// TwinCAT 3 PLC project PLC1
// ProgramVersion: 3.1.4026.16
// CompilerDefines: VISU_USEPROPERTYINFO
// libraries:
//   SH_Light, * (StroemHansen)
//   Tc2_EnOcean, * (Beckhoff Automation GmbH)
//   Tc2_Standard, * (Beckhoff Automation GmbH)
//   Tc2_System, * (Beckhoff Automation GmbH)
//   Tc2_Utilities, * (Beckhoff Automation GmbH)
//   Tc3_DALI, * (Beckhoff Automation GmbH)
//   Tc3_System_DK, * (Beckhoff - DK)
//   VisuDialogs, * (System)
// project tree:
//   DUTs/DALI/ E_DALIExtendedFadeTime.TcTLEO (not stored), ST_DALI102Parameters.TcDUT (not stored), ST_DALI103Parameters.TcDUT (not stored), ST_DALIMemoryBank.TcDUT (not stored), ST_DALI_GrpAssignment.TcDUT (not stored), ST_GroupSort.TcDUT (not stored)
//   DUTs/EnOcean/ ST_ReadSAB05.TcDUT (not stored), ST_WriteSAB05.TcDUT (not stored)
//   / FastTask.TcTTO (not stored), GlobalTextList.TcGTLO (not stored), PlcTask.TcTTO (not stored), Visualization Manager.TcVMO (not stored)
//   GVLs/ GVL_AHDataModbus.TcGVL, GVL_EnOcean.TcGVL, GVL_Skalering.TcGVL
//   POUs/01_System/01_System/GVLs/ GVL_EtherCAT.TcGVL (not stored)
//   POUs/01_System/01_System/ P_SystemDK.TcPOU (not stored)
//   POUs/AHModbusComm/ P_AHModbusComm.TcPOU
//   POUs/Alle_Rum/Gange/Gang_3_109/ P_Gang_3_109_Kantine.TcPOU, Visualization_4_308.TcVIS (excluded from build)
//   POUs/Alle_Rum/Gange/Gang_4_208/ P_Gang_4_208.TcPOU, Visualization_5_338_1.TcVIS (excluded from build)
//   POUs/Alle_Rum/Gange/Gang_4_211/ P_Gang_4_211.TcPOU, Visualization_5_338_1_1_1_1.TcVIS (excluded from build)
//   POUs/Alle_Rum/Gange/Gang_4_210A/ P_Gang_4_210A.TcPOU, Visualization_4_307_1_1.TcVIS (excluded from build)
//   POUs/Alle_Rum/Rum_Med_DALI_Pir/Rum_4_206/ P_Rum_4_206.TcPOU, Visualization_5_338_1_1.TcVIS (excluded from build)
//   POUs/Alle_Rum/Rum_Med_DALI_Pir/Rum_4_211A/ P_Rum_4_211A.TcPOU, Visualization_5_338_1_1_1.TcVIS (excluded from build)
//   POUs/Alle_Rum/Rum_Med_DALI_Pir/Rum_4_207/ P_Rum_4_207.TcPOU, Visualization_4_307_1.TcVIS (excluded from build)
//   POUs/Alle_Rum/Rum_Med_DALI_Pir/Rum_4_213_Og_4_215_Foldedoer/ P_Foldedoer_4_213.TcPOU, P_Rum_4_213.TcPOU, P_Rum_4_215.TcPOU
//   POUs/Alle_Rum/Trapper/ P_DigTest.TcPOU
//   POUs/DALI/DALI_Setup/ DALI_Commissioning.TcPOU (not stored)
//   POUs/DALI/DALI_Setup/FBs/ FB_Part102Addressing.TcPOU (not stored), FB_Part102Commands.TcPOU (not stored), FB_Part102Groups.TcPOU (not stored), FB_Part102MemoryPages.TcPOU (not stored), FB_Part102Parameters.TcPOU (not stored), FB_Part102Scenes.TcPOU (not stored), FB_Part102SetFading.TcPOU (not stored), FB_Part103Addressing.TcPOU (not stored), FB_Part103MemoryPages.TcPOU (not stored), FB_Part103Identify.TcPOU (not stored), FB_Part103Parameters.TcPOU (not stored), FB_Part202Emergency.TcPOU (not stored), FB_Part205Incandescent.TcPOU (not stored), FB_Part207LED.TcPOU (not stored), FB_Part208Switching.TcPOU (not stored), FB_Part300GenericDevice.TcPOU (not stored), FB_Part301PushButton.TcPOU (not stored), FB_Part302AbsoluteInputDevice.TcPOU (not stored), FB_Part303OccupancySensor.TcPOU (not stored), FB_Part304LightSensor.TcPOU (not stored), GearType.TcPOU (not stored)
//   POUs/DALI/DALI_Setup/GVLs/ GVL_Internal.TcGVL (not stored)
//   POUs/DALI/DALI_Setup/VISUs/TextLists/ CommandOnTerminalEvent.TcTLO, DimmingCurve.TcTLO, EventPriority.TcTLO (not stored), EventScheme.TcTLO, ExtendedFadeTime.TcTLO (not stored), FadeRate.TcTLO (not stored), FadeTime.TcTLO, FastFadeTime.TcTLO (not stored), TextList_Dialogs.TcTLO (not stored)
//   POUs/DALI/DALI_Setup/VISUs/ Visu_DALICommissioning.TcVIS
//   POUs/DALI/DALI_Setup/VISUs/Visu_DALICommissioning/ Visu_KL6821Configuration.TcVIS (not stored) (excluded from build), Visu_Part102Addressing.TcVIS, Visu_Part102Commands.TcVIS (not stored), Visu_Part102Groups.TcVIS, Visu_Part102MemoryBank.TcVIS (not stored), Visu_Part102Parameters.TcVIS, Visu_Part102Scenes.TcVIS, Visu_Part102SetFading.TcVIS, Visu_Part103Addressing.TcVIS, Visu_Part103Identify.TcVIS (not stored), Visu_Part103MemoryBank.TcVIS (not stored), Visu_Part103Parameters.TcVIS (not stored), Visu_Part202.TcVIS (not stored), Visu_Part202Commands.TcVIS (not stored), Visu_Part202Parameters.TcVIS (not stored), Visu_Part202Status.TcVIS (not stored), Visu_Part205.TcVIS (not stored), Visu_Part205Parameters.TcVIS (not stored), Visu_Part205Status.TcVIS (not stored), Visu_Part207.TcVIS, Visu_Part207Parameters.TcVIS (not stored), Visu_Part207Status.TcVIS, Visu_Part208Switching.TcVIS (not stored), Visu_Part300GenericDevice.TcVIS, Visu_Part301PushButton.TcVIS (not stored), Visu_Part302AbsoluteInputDevice.TcVIS (not stored), Visu_Part303OccupancySensor.TcVIS, Visu_Part304LightSensor.TcVIS (not stored), Visu_Welcome.TcVIS (not stored)
//   POUs/DALI/PRGs/Background/ P_DALI_Background.TcPOU (not stored)
//   POUs/DALI/PRGs/Diag/ P_DALI_DIAG.TcPOU (not stored)
//   POUs/DALI/PRGs/EnergyData/ P_DALI_Energy_Firmware_Test.TcPOU (not stored) (excluded from build), P_DALI_Energy_Line.TcPOU (not stored)
//   POUs/EnOcean/ P_EnOcean.TcPOU
//   POUs/ MAIN.TcPOU
//   POUs/Tester/ P_DALI2_Test.TcPOU (not stored) (excluded from build), P_Test_TypeA.TcPOU (not stored) (excluded from build), Visualization.TcVIS (not stored) (excluded from build)
// real-time tasks:
//   TASK PlcTask: cycle T#40ms, priority 21, ADS port 350
//   TASK FastTask: cycle T#4ms, priority 20, ADS port 351
// I/O:
//   DEVICE Device 1 (Beckhoff CCAT)
//   DEVICE Device 3 (CX-BK)
//     Box 1 (CX-BK)
// variable links:
//   PLC1/PLC1 Instance <-> Device 3 (CX-BK)/Box 1 (CX-BK)
//     FastTask Inputs/P_DALI_Background.arrKL6821InData[1] @bit 16 <-> Term 4 (KL6821)/Channel 1/Data In 0
//     FastTask Inputs/P_DALI_Background.arrKL6821InData[1] @bit 24 <-> Term 4 (KL6821)/Channel 1/Data In 1
//     FastTask Inputs/P_DALI_Background.arrKL6821InData[1] @bit 32 <-> Term 4 (KL6821)/Channel 1/Data In 2
//     FastTask Inputs/P_DALI_Background.arrKL6821InData[1] @bit 40 <-> Term 4 (KL6821)/Channel 1/Data In 3
//     FastTask Inputs/P_DALI_Background.arrKL6821InData[2] @bit 16 <-> Term 5 (KL6821)/Channel 1/Data In 0
//     FastTask Inputs/P_DALI_Background.arrKL6821InData[2] @bit 24 <-> Term 5 (KL6821)/Channel 1/Data In 1
//     FastTask Inputs/P_DALI_Background.arrKL6821InData[2] @bit 32 <-> Term 5 (KL6821)/Channel 1/Data In 2
//     FastTask Inputs/P_DALI_Background.arrKL6821InData[2] @bit 40 <-> Term 5 (KL6821)/Channel 1/Data In 3
//     FastTask Inputs/P_DALI_Background.arrKL6821InData[3] @bit 16 <-> Term 6 (KL6821)/Channel 1/Data In 0
//     FastTask Inputs/P_DALI_Background.arrKL6821InData[3] @bit 24 <-> Term 6 (KL6821)/Channel 1/Data In 1
//     FastTask Inputs/P_DALI_Background.arrKL6821InData[3] @bit 32 <-> Term 6 (KL6821)/Channel 1/Data In 2
//     FastTask Inputs/P_DALI_Background.arrKL6821InData[3] @bit 40 <-> Term 6 (KL6821)/Channel 1/Data In 3
//     FastTask Inputs/P_DALI_Background.arrKL6821InData[1] <-> Term 4 (KL6821)/Channel 1/State
//     FastTask Inputs/P_DALI_Background.arrKL6821InData[2] <-> Term 5 (KL6821)/Channel 1/State
//     FastTask Inputs/P_DALI_Background.arrKL6821InData[3] <-> Term 6 (KL6821)/Channel 1/State
//     FastTask Inputs/P_EnOcean.stKL6581_in @bit 8 <-> Term 2 (KL6581)/Channel 1/Input CNODE
//     FastTask Inputs/P_EnOcean.stKL6581_in @bit {24..48 step 8} <-> Term 2 (KL6581)/Channel 1/Input DB{0..3}  (4 links)
//     FastTask Inputs/P_EnOcean.stKL6581_in @bit {56..80 step 8} <-> Term 2 (KL6581)/Channel 1/Input ID{0..3}  (4 links)
//     FastTask Inputs/P_EnOcean.stKL6581_in @bit 16 <-> Term 2 (KL6581)/Channel 1/Input ORG
//     FastTask Inputs/P_EnOcean.stKL6581_in @bit 88 <-> Term 2 (KL6581)/Channel 1/Input STATUS
//     FastTask Inputs/P_EnOcean.stKL6581_in <-> Term 2 (KL6581)/Channel 1/Status
//     FastTask Outputs/P_DALI_Background.arrKL6821OutData[1] <-> Term 4 (KL6821)/Channel 1/Ctrl
//     FastTask Outputs/P_DALI_Background.arrKL6821OutData[2] <-> Term 5 (KL6821)/Channel 1/Ctrl
//     FastTask Outputs/P_DALI_Background.arrKL6821OutData[3] <-> Term 6 (KL6821)/Channel 1/Ctrl
//     FastTask Outputs/P_DALI_Background.arrKL6821OutData[1] @bit 16 <-> Term 4 (KL6821)/Channel 1/Data Out 0
//     FastTask Outputs/P_DALI_Background.arrKL6821OutData[1] @bit 24 <-> Term 4 (KL6821)/Channel 1/Data Out 1
//     FastTask Outputs/P_DALI_Background.arrKL6821OutData[1] @bit 32 <-> Term 4 (KL6821)/Channel 1/Data Out 2
//     FastTask Outputs/P_DALI_Background.arrKL6821OutData[1] @bit 40 <-> Term 4 (KL6821)/Channel 1/Data Out 3
//     FastTask Outputs/P_DALI_Background.arrKL6821OutData[2] @bit 16 <-> Term 5 (KL6821)/Channel 1/Data Out 0
//     FastTask Outputs/P_DALI_Background.arrKL6821OutData[2] @bit 24 <-> Term 5 (KL6821)/Channel 1/Data Out 1
//     FastTask Outputs/P_DALI_Background.arrKL6821OutData[2] @bit 32 <-> Term 5 (KL6821)/Channel 1/Data Out 2
//     FastTask Outputs/P_DALI_Background.arrKL6821OutData[2] @bit 40 <-> Term 5 (KL6821)/Channel 1/Data Out 3
//     FastTask Outputs/P_DALI_Background.arrKL6821OutData[3] @bit 16 <-> Term 6 (KL6821)/Channel 1/Data Out 0
//     FastTask Outputs/P_DALI_Background.arrKL6821OutData[3] @bit 24 <-> Term 6 (KL6821)/Channel 1/Data Out 1
//     FastTask Outputs/P_DALI_Background.arrKL6821OutData[3] @bit 32 <-> Term 6 (KL6821)/Channel 1/Data Out 2
//     FastTask Outputs/P_DALI_Background.arrKL6821OutData[3] @bit 40 <-> Term 6 (KL6821)/Channel 1/Data Out 3
//     FastTask Outputs/P_EnOcean.stKL6581_out <-> Term 2 (KL6581)/Channel 1/Control
//     FastTask Outputs/P_EnOcean.stKL6581_out @bit 8 <-> Term 2 (KL6581)/Channel 1/Output CNODE
//     FastTask Outputs/P_EnOcean.stKL6581_out @bit {24..48 step 8} <-> Term 2 (KL6581)/Channel 1/Output DB{0..3}  (4 links)
//     FastTask Outputs/P_EnOcean.stKL6581_out @bit {56..80 step 8} <-> Term 2 (KL6581)/Channel 1/Output ID{0..3}  (4 links)
//     FastTask Outputs/P_EnOcean.stKL6581_out @bit 16 <-> Term 2 (KL6581)/Channel 1/Output ORG
//     FastTask Outputs/P_EnOcean.stKL6581_out @bit 88 <-> Term 2 (KL6581)/Channel 1/Output STATUS
//     PlcTask Inputs/MAIN.nCX8200_State <-> Inputs/State
//     PlcTask Inputs/P_Foldedoer_4_213.bFoldingDoorOpen <-> Term 3 (KL1408)/Channel 2/Input

// ---- GVLs/GVL_AHDataModbus.TcGVL
{attribute 'qualified_only'}
VAR_GLOBAL
//AH pir data out
	nAH_NeighborRoomsPir_Out		    AT %MB600	: UINT;
	
//AH pir data in
	arrAH_NeighborRoomsPir_In								: ARRAY[1..byNumberOfAH_Neighbors] OF UINT;
	arrAH_NeighborRoomsPir										: ARRAY[1..byNumberOfAH_Neighbors] OF ARRAY[0..15] OF BOOL;
	
//Schneider data out
	nCX8200_State_MB					AT %MB1000		: UINT;
	arrFB_DALIDiagErrorId			(*AT %MW1002*)	: ARRAY[1..SH_Light.DALI_Param.MAX_DALIV2_LINES] OF UDINT;
	arrKL6821InDataStatus				AT %MB1014		: ARRAY[1..SH_Light.DALI_Param.MAX_DALIV2_LINES] OF WORD;
	arrDALILineShrtAddrErr				AT %MB1026		: ARRAY[1..SH_Light.DALI_Param.MAX_DALIV2_LINES] OF UINT;
	EnOceanError						AT %MB1038		: UINT;
	nTotalEnergy10kWh						AT %MB1040		: UINT;
	nMaxControlGearOperatingHours 	    AT %MB1042		: UINT;
		uiPirOffDelayTimeAllRooms_MB   AT %MB1044   : UINT := 30;
END_VAR
VAR_GLOBAL CONSTANT
	byNumberOfAH_Neighbors									: BYTE := 25;
END_VAR

// ---- GVLs/GVL_EnOcean.TcGVL
{attribute 'qualified_only'}
VAR_GLOBAL
//Atrium
	strEnOceanSwitch_Gang_3_109_PladeA				: Tc2_EnOcean.STR_EnOceanSwitch;
	strEnOceanSwitch_AtriumNiveau_PladeB				: Tc2_EnOcean.STR_EnOceanSwitch;
	strEnOceanSwitch_AtriumNiveau_Service				: Tc2_EnOcean.STR_EnOceanSwitch;	

	//Gange
    strEnOceanSwitch_Gang_4_211_Indgang				: Tc2_EnOcean.STR_EnOceanSwitch;
	strEnOceanSwitch_Gang_4_211_Ekstra					: Tc2_EnOcean.STR_EnOceanSwitch;
	
	//Rum				
	strEnOceanSwitch_Rum_4_206_Indgang				: Tc2_EnOcean.STR_EnOceanSwitch;
	strEnOceanSwitch_Rum_4_206_Ekstra					: Tc2_EnOcean.STR_EnOceanSwitch;
	
	strEnOceanSwitch_Rum_4_207_Indgang				: Tc2_EnOcean.STR_EnOceanSwitch;
	strEnOceanSwitch_Rum_4_207_Ekstra					: Tc2_EnOcean.STR_EnOceanSwitch;
	
	strEnOceanSwitch_Rum_4_211A_Indgang				: Tc2_EnOcean.STR_EnOceanSwitch;
	strEnOceanSwitch_Rum_4_211A_Ekstra				: Tc2_EnOcean.STR_EnOceanSwitch;
	
	strEnOceanSwitch_Rum_4_213_Indgang				: Tc2_EnOcean.STR_EnOceanSwitch;
	strEnOceanSwitch_Rum_4_213_Pendler				: Tc2_EnOcean.STR_EnOceanSwitch;
	
	strEnOceanSwitch_Rum_4_215								: Tc2_EnOcean.STR_EnOceanSwitch;
	
END_VAR

// ---- GVLs/GVL_Skalering.TcGVL
//{attribute 'qualified_only'}
VAR_GLOBAL
rMeassure_Zone1 :REAL:= 604; 
rRead_Zone1     :REAL:= 340;

rMeassure_Zone2 :REAL:=611;
rRead_Zone2     :REAL:=374;

rMeassure_Zone3 :REAL:=986;
rRead_Zone3     :REAL:=524;

rMeassure_Zone4 :REAL:=770;
rRead_Zone4     :REAL:=506;

rMeassure_Zone5 :REAL:=734;
rRead_Zone5     :REAL:=395;

rMeassure_Zone6 :REAL:=890;
rRead_Zone6     :REAL:=476;

rMeassure_Zone7 :REAL:=710;
rRead_Zone7     :REAL:=654;

rMeassure_Zone8 :REAL:=604;
rRead_Zone8     :REAL:=292;

rMeassure_Zone9 :REAL:=572;
rRead_Zone9     :REAL:=348;

rMeassure_Zone10:REAL:= 790;
rRead_Zone10    :REAL:=434;

rMeassure_Zone11 :REAL:=691;
rRead_Zone11     :REAL:=426;

END_VAR

// ---- POUs/AHModbusComm/P_AHModbusComm.TcPOU
PROGRAM P_AHModbusComm
VAR
	arrfbReadAHPirData		: ARRAY[1..GVL_AHDataModbus.byNumberOfAH_Neighbors] OF SH_Light.FB_ReadAHPirData;
	arrReadAHPirData			: ARRAY[1..GVL_AHDataModbus.byNumberOfAH_Neighbors] OF BOOL;
	
	arrfbTriggerPulses			: ARRAY[1..GVL_AHDataModbus.byNumberOfAH_Neighbors] OF SH_Light.FB_ClockPulse;
	arrGeneratePulses			: ARRAY[1..GVL_AHDataModbus.byNumberOfAH_Neighbors] OF BOOL := [GVL_AHDataModbus.byNumberOfAH_Neighbors(TRUE)];
	tTimeInterval					: TIME := T#1S;
	tPulseTime					: TIME := T#1S;
	
	byLineId						: BYTE;
	byAHId							: BYTE;
	
			
	fbWritePirDelayTime		: R_TRIG;
	bRunOverrideOnce		: BOOL := FALSE;
	bEnableDelayTimeOverride : BOOL := FALSE;
	uiPirOffDelayTimeAllRooms : UINT := 30;
END_VAR

VAR CONSTANT
	arrstNeighborIPAddr					: ARRAY[1..GVL_AHDataModbus.byNumberOfAH_Neighbors] OF SH_Light.ST_NeighborIP := [
																								(sIP := '172.24.195.161', IsNeighbor := FALSE),
																							    (sIP := '172.24.195.162', IsNeighbor := FALSE), // AH1-2
																								(sIP := '172.24.195.163', IsNeighbor := FALSE), 
																							(sIP := '172.24.195.164', IsNeighbor := TRUE), 
																							(sIP := '172.24.195.165', IsNeighbor := TRUE), 
																								(sIP := '172.24.195.166', IsNeighbor := FALSE), 
																								(sIP := '172.24.195.167', IsNeighbor := FALSE), 
																								(sIP := '172.24.195.168', IsNeighbor := FALSE), 
																							(sIP := '172.24.195.169', IsNeighbor := TRUE), // AH3-2
																								(sIP := '172.24.195.170', IsNeighbor := FALSE), 
																								(sIP := '172.24.195.171', IsNeighbor := FALSE), 
																								(sIP := '172.24.195.172', IsNeighbor := FALSE), 
																								(sIP := '172.24.195.173', IsNeighbor := FALSE), 
																							(sIP := '172.24.195.174', IsNeighbor := TRUE), 
																								(sIP := '172.24.195.175', IsNeighbor := FALSE), 
																								(sIP := '172.24.195.176', IsNeighbor := FALSE), 
																								(sIP := '172.24.195.177', IsNeighbor := FALSE),
																							(sIP := '172.24.195.178', IsNeighbor := TRUE),
																							(sIP := '172.24.195.179', IsNeighbor := TRUE), // AH5-2
																								(sIP := '172.24.195.180', IsNeighbor := FALSE),
																								(sIP := '172.24.195.181', IsNeighbor := FALSE),
																								(sIP := '172.24.195.182', IsNeighbor := FALSE),
																								(sIP := '172.24.195.183', IsNeighbor := FALSE),
																								(sIP := '172.24.195.184', IsNeighbor := FALSE),
																								(sIP := '172.24.195.185', IsNeighbor := FALSE)];
	arrMBAddr					: ARRAY[1..GVL_AHDataModbus.byNumberOfAH_Neighbors] OF WORD := [GVL_AHDataModbus.byNumberOfAH_Neighbors(12588)]; //modbus-adresser
END_VAR

A_AHNeighborRoomsPirIn();
A_AHNeighborRoomsPirOut();
A_DALILineShrtAddrErr();
A_DelayTimeAllRooms();

ACTION A_AHNeighborRoomsPirIn:
FOR byAHId := 1 TO GVL_AHDataModbus.byNumberOfAH_Neighbors DO
//Generate Pulses
	arrfbTriggerPulses[byAHId](bGenerateClockPulses:= arrGeneratePulses[byAHId], tTimeInterval:= tTimeInterval, tPulseTime:= tPulseTime);
	arrReadAHPirData[byAHId]:= arrfbTriggerPulses[byAHId].bPulse;
//Read data
	IF arrstNeighborIPAddr[byAHId].IsNeighbor THEN
	arrfbReadAHPirData[byAHId](	bReadAHPirData			:=	arrReadAHPirData[byAHId],
													sIPAddr							:=	arrstNeighborIPAddr[byAHId].sIP,
													nMBAddr						:=	arrMBAddr[byAHId],
													nMBDataBuffer				:=	GVL_AHDataModbus.arrAH_NeighborRoomsPir_In[byAHId],
													arrAH_NeighborRoomsPir	=>GVL_AHDataModbus.arrAH_NeighborRoomsPir[byAHId]);
	END_IF
END_FOR
END_ACTION

ACTION A_AHNeighborRoomsPirOut:
GVL_AHDataModbus.nAH_NeighborRoomsPir_Out.0		:= P_Gang_3_109_Kantine.bPirActive_MB;
GVL_AHDataModbus.nAH_NeighborRoomsPir_Out.1		:= P_Gang_4_208.bPirActive_MB;
//GVL_AHDataModbus.nAH_NeighborRoomsPir_Out.2		:=
//GVL_AHDataModbus.nAH_NeighborRoomsPir_Out.3		:=
//GVL_AHDataModbus.nAH_NeighborRoomsPir_Out.4		:= 
//GVL_AHDataModbus.nAH_NeighborRoomsPir_Out.5		:= 
//GVL_AHDataModbus.nAH_NeighborRoomsPir_Out.6		:=
//GVL_AHDataModbus.nAH_NeighborRoomsPir_Out.7		:= 
//GVL_AHDataModbus.nAH_NeighborRoomsPir_Out.8		:=
//GVL_AHDataModbus.nAH_NeighborRoomsPir_Out.9		:= 
//GVL_AHDataModbus.nAH_NeighborRoomsPir_Out.10	:
//GVL_AHDataModbus.nAH_NeighborRoomsPir_Out.11	:= 
//GVL_AHDataModbus.nAH_NeighborRoomsPir_Out.12	:=
//GVL_AHDataModbus.nAH_NeighborRoomsPir_Out.13	:=
END_ACTION

ACTION A_DALILineShrtAddrErr:
FOR  byLineId := 1 TO SH_Light.DALI_Param.MAX_DALIV2_LINES DO
	GVL_AHDataModbus.arrDALILineShrtAddrErr[byLineId] :=  TO_UINT(SH_Light.GVL_DALI_LatestError.arrLineShrtAddr[byLineId]);
END_FOR
END_ACTION

ACTION A_DelayTimeAllRooms:

fbWritePirDelayTime(CLK := GVL_AHDataModbus.uiPirOffDelayTimeAllRooms_MB<>uiPirOffDelayTimeAllRooms);

IF fbWritePirDelayTime.Q THEN
	bRunOverrideOnce := TRUE;
	bEnableDelayTimeOverride := TRUE;
	
//Indsæt kode
P_Gang_3_109_Kantine.fbWritePirDelayTIme(bEnableOverride := bEnableDelayTimeOverride, nOverRideValue := GVL_AHDataModbus.uiPirOffDelayTimeAllRooms_MB, nValIn1 := GVL_AHDataModbus.uiPirOffDelayTimeAllRooms_MB, nValIn2 := uiPirOffDelayTimeAllRooms);
P_Gang_4_208.fbWritePirDelayTIme(bEnableOverride := bEnableDelayTimeOverride, nOverRideValue := GVL_AHDataModbus.uiPirOffDelayTimeAllRooms_MB, nValIn1 := GVL_AHDataModbus.uiPirOffDelayTimeAllRooms_MB, nValIn2 := uiPirOffDelayTimeAllRooms);
P_Rum_4_206.fbWritePirDelayTIme(bEnableOverride := bEnableDelayTimeOverride, nOverRideValue := GVL_AHDataModbus.uiPirOffDelayTimeAllRooms_MB, nValIn1 := GVL_AHDataModbus.uiPirOffDelayTimeAllRooms_MB, nValIn2 := uiPirOffDelayTimeAllRooms);
P_Rum_4_207.fbWritePirDelayTIme(bEnableOverride := bEnableDelayTimeOverride, nOverRideValue := GVL_AHDataModbus.uiPirOffDelayTimeAllRooms_MB, nValIn1 := GVL_AHDataModbus.uiPirOffDelayTimeAllRooms_MB, nValIn2 := uiPirOffDelayTimeAllRooms);
P_Rum_4_211A.fbWritePirDelayTIme(bEnableOverride := bEnableDelayTimeOverride, nOverRideValue := GVL_AHDataModbus.uiPirOffDelayTimeAllRooms_MB, nValIn1 := GVL_AHDataModbus.uiPirOffDelayTimeAllRooms_MB, nValIn2 := uiPirOffDelayTimeAllRooms);
P_Rum_4_213.fbWritePirDelayTIme(bEnableOverride := bEnableDelayTimeOverride, nOverRideValue := GVL_AHDataModbus.uiPirOffDelayTimeAllRooms_MB, nValIn1 := GVL_AHDataModbus.uiPirOffDelayTimeAllRooms_MB, nValIn2 := uiPirOffDelayTimeAllRooms);
P_Gang_4_211.fbWritePirDelayTIme(bEnableOverride := bEnableDelayTimeOverride, nOverRideValue := GVL_AHDataModbus.uiPirOffDelayTimeAllRooms_MB, nValIn1 := GVL_AHDataModbus.uiPirOffDelayTimeAllRooms_MB, nValIn2 := uiPirOffDelayTimeAllRooms);
P_Rum_4_215.fbWritePirDelayTIme(bEnableOverride := bEnableDelayTimeOverride, nOverRideValue := GVL_AHDataModbus.uiPirOffDelayTimeAllRooms_MB, nValIn1 := GVL_AHDataModbus.uiPirOffDelayTimeAllRooms_MB, nValIn2 := uiPirOffDelayTimeAllRooms);ELSE
	IF bRunOverrideOnce THEN
		bEnableDelayTimeOverride := FALSE;
		
		//Indsæt kode
P_Gang_3_109_Kantine.fbWritePirDelayTIme(bEnableOverride := bEnableDelayTimeOverride, nOverRideValue := GVL_AHDataModbus.uiPirOffDelayTimeAllRooms_MB, nValIn1 := GVL_AHDataModbus.uiPirOffDelayTimeAllRooms_MB, nValIn2 := uiPirOffDelayTimeAllRooms);
P_Gang_4_208.fbWritePirDelayTIme(bEnableOverride := bEnableDelayTimeOverride, nOverRideValue := GVL_AHDataModbus.uiPirOffDelayTimeAllRooms_MB, nValIn1 := GVL_AHDataModbus.uiPirOffDelayTimeAllRooms_MB, nValIn2 := uiPirOffDelayTimeAllRooms);
P_Rum_4_206.fbWritePirDelayTIme(bEnableOverride := bEnableDelayTimeOverride, nOverRideValue := GVL_AHDataModbus.uiPirOffDelayTimeAllRooms_MB, nValIn1 := GVL_AHDataModbus.uiPirOffDelayTimeAllRooms_MB, nValIn2 := uiPirOffDelayTimeAllRooms);
P_Rum_4_207.fbWritePirDelayTIme(bEnableOverride := bEnableDelayTimeOverride, nOverRideValue := GVL_AHDataModbus.uiPirOffDelayTimeAllRooms_MB, nValIn1 := GVL_AHDataModbus.uiPirOffDelayTimeAllRooms_MB, nValIn2 := uiPirOffDelayTimeAllRooms);
P_Rum_4_211A.fbWritePirDelayTIme(bEnableOverride := bEnableDelayTimeOverride, nOverRideValue := GVL_AHDataModbus.uiPirOffDelayTimeAllRooms_MB, nValIn1 := GVL_AHDataModbus.uiPirOffDelayTimeAllRooms_MB, nValIn2 := uiPirOffDelayTimeAllRooms);
P_Rum_4_213.fbWritePirDelayTIme(bEnableOverride := bEnableDelayTimeOverride, nOverRideValue := GVL_AHDataModbus.uiPirOffDelayTimeAllRooms_MB, nValIn1 := GVL_AHDataModbus.uiPirOffDelayTimeAllRooms_MB, nValIn2 := uiPirOffDelayTimeAllRooms);
P_Gang_4_211.fbWritePirDelayTIme(bEnableOverride := bEnableDelayTimeOverride, nOverRideValue := GVL_AHDataModbus.uiPirOffDelayTimeAllRooms_MB, nValIn1 := GVL_AHDataModbus.uiPirOffDelayTimeAllRooms_MB, nValIn2 := uiPirOffDelayTimeAllRooms);
P_Rum_4_215.fbWritePirDelayTIme(bEnableOverride := bEnableDelayTimeOverride, nOverRideValue := GVL_AHDataModbus.uiPirOffDelayTimeAllRooms_MB, nValIn1 := GVL_AHDataModbus.uiPirOffDelayTimeAllRooms_MB, nValIn2 := uiPirOffDelayTimeAllRooms);



bRunOverrideOnce := FALSE;
	END_IF
END_IF
END_ACTION

END_PROGRAM

// ---- POUs/Alle_Rum/Gange/Gang_3_109/P_Gang_3_109_Kantine.TcPOU
PROGRAM P_Gang_3_109_Kantine
VAR
(*Gangen består af to lysgrupper - 5 og 14 - på to forskellige DALI-linjer - 2 og 1 henh..
Begge grupper afhænger af samme PIR-input - pir-adr. 6, 7, 8, 9 og 10 - på DALI-linje 2.
Derfor oprettes to adskilte reguleringer med samme PV. Dvs., at knapfunktion og pirfunktion forbliver den samme.

En anden del af af hele gangen styres fra AH4_3. De to dele nabostyres med PIR-signaler over modbus-kommunikation*)

	arrfbLysGruppe			: ARRAY [1..2] OF FB_Light_Type_B;
	arrstDaliSetupGruppe	: ARRAY[1..2] OF SH_Light.ST_DALI_RoomSetup := 
	
													[(	byShrtAdr_Prim := 26, 
														byGrpAdr_Prim := 6, 
														eMod_Prim := E_DALIAddressType.Group, 
														//byShrtAdr_Sec := 1, 
														//byGrpAdr_Sec := 1, 
														//eMod_Sec := E_DALIAddressType.Short, 
														//byShrtAdr_Supl := 1, 
														DALI_LINE_NUM_PRIM := arrDALI_LINE_NUM_LIGHT[1], 
														DALI_LINE_NUM_SEC := 0, //0 = ingen zonestyring/vinduerække
														DALI_LINE_NUM_SUPL := arrDALI_LINE_NUM_PENDANTS[1]),
														
													(	byShrtAdr_Prim := 31, 
														byGrpAdr_Prim := 6, 
														eMod_Prim := E_DALIAddressType.Group, 
														//byShrtAdr_Sec := 1, 
														//byGrpAdr_Sec := 1, 
														//eMod_Sec := E_DALIAddressType.Short, 
														//byShrtAdr_Supl := 1, 
														DALI_LINE_NUM_PRIM := arrDALI_LINE_NUM_LIGHT[2], 
														DALI_LINE_NUM_SEC := 0, 
														DALI_LINE_NUM_SUPL := arrDALI_LINE_NUM_PENDANTS[2])];
														
	arrstLiveDataGruppe		: ARRAY [1..2] OF SH_Light.ST_LiveData;
	//stLiveData AT %MB22	: SH_Light.ST_LiveData;
	
	arrRunTuningGruppe: ARRAY[1..2] OF BOOL;
	
	
	
	bTopButtonZone1			: BOOL;
	bTopButtonZone1_Visu	: BOOL;
	bBottomButtonZone1		: BOOL;
	bBottomButtonZone1_Visu	: BOOL;
	bButtonZone2			: BOOL;
	bNeighborRoomsPir		: BOOL;
	fLuxOn					: REAL;
	fLuxDim					: REAL;
	tPIRDim					: TIME;
	tPIROff					: TIME;
	fOffsetSec				: REAL := 20;
	bOccupiedRoom			: BOOL;

	bRunTuning				: BOOL;
	


// Sensor Settings
	//fbSensor					: SH_Light.FB_NIKO_P46xx_1Pcs;
	fbSensor					: SH_Light.FB_NIKO_P46xx_3Pcs;
	//bySensorAddr				: BYTE := 17;
	arrSensorAddr				: ARRAY[1..3] OF BYTE := [3,4,5];
	bInitialize					: BOOL := TRUE;
	stDaliSensorSetup			: ST_DALI_NIKOP46SetupData;
	//bInitErr					: BOOL;
	//bInitDone					: BOOL;
	arrInitErr					: ARRAY [1..3] OF BOOL;
	arrInitDone					: ARRAY [1..3] OF BOOL;
	arrSensorScales				: ARRAY [1..10] OF SH_Light.ST_DALI_SensorScaleMode := [	(fMeassureMaxSensor := rMeassure_Zone11, fReadMaxSensor := rRead_Zone11),
																							(fMeassureMaxSensor := rMeassure_Zone11, fReadMaxSensor := rRead_Zone11),
																							(fMeassureMaxSensor := rMeassure_Zone11, fReadMaxSensor := rRead_Zone11),																					
																						7(())];
	bCancelHoldTimerOccupancy	: BOOL;
(*	eEventPriorityOccupancy		: E_DALIEventPriority := E_DALIEVENTPRIORITY.Middle;
	nHoldTimerOccupancy			: WORD := 5; // Value in s. 	
	nReportTimerOccupancy		: BYTE := 120; // Value in s, Preset manufacturer value
	nDeadtimeTimerOccupancy		: WORD := 100; // Value in ms, Predefined Value of DALI Standard
	bCancelHoldTimerOccupancy	: BOOL;
	nSensitivityOccupancy		: BYTE:= 3; //setting Sensivity (0..4) 0 (Off), 1 (Min), 2(Low), 3(High) and 4 (Max)

	bEnableLuxEvent				: BOOL;
	eEventPriorityBrightness	: E_DALIEventPriority := E_DALIEVENTPRIORITY.Middle;
	nDeadtimeTimerBrightness	: WORD := 1500; // Value in ms, Predefined Value of DALI Standard
	nHysteresisBrightness		: BYTE := 2; // Value in %
	nHysteresisMinBrightness	: BYTE := 10; // Absolute Value, depending on the manufacturer specific resolution
	nReportTimerBrightness		: BYTE := 120; // Value in s, Preset manufacturer value
*)

	//ModbusComm setup
	
	fbWriteSPLuxLevel			: SH_Light.FB_TwoVal_SelectOne_RTrigChange;
	fbWritePirDelayTIme			: SH_Light.FB_TwoVal_SelectOne_RTrigChange;
	stRoomDataPLC				: SH_Light.ST_RoomDataPLC	:=	(	uiPirOffDelayTime	:= 30,
																	uiSpLuxLevel		:= 500,
																	uiPirDimDelayTime	:= 15,
																	uiSpDimLuxLevel		:= 200
																);
	fbBallastOnHours			: SH_Light.FB_CountOnHours;
	bEnableHourCount			: BOOL := TRUE;
	
	//Non-persistent modbus data
	bPirActive_MB			AT%MX0.0	: BOOL;				//bPirLys i gammel kode
	uiActLuxLevel_MB		AT%MB4					: UINT;				//intHMIAktueltLux i gammel kode
	uiActLightLevelPct_MB	AT%MB10					: UINT;				//intDALI_Gruppe1_Lysniveau i gammel kode
	
	//For Conversion
	uiPirOffMinutes						: UINT;
	udTimeScaling						: UDINT := 60000;
	uiLuxOn								: UINT;
	
	//max values checks
	uiMaxLuxLevel						: UINT := 1023;
	uiMaxPirOffMinutes					: UINT := 180;

END_VAR

VAR CONSTANT
	Sensor_DALI_LINE_NUM: BYTE := 1;
	arrDALI_LINE_NUM_LIGHT: ARRAY[1..2] OF BYTE := [2,1]; //korrekt rækkefølge nødvendig
	arrDALI_LINE_NUM_PENDANTS: ARRAY[1..2] OF BYTE := [0,0]; //korrekt rækkefølge nødvendig. 0 = ingen pendler
END_VAR
VAR PERSISTENT
	stPirSensorData: SH_Light.ST_DALI_Sensor;
	arrstTuneDataGruppe: ARRAY [1..2] OF SH_Light.ST_TuneData_EX;
	
	uiPirOffDelayTime_MB	AT %MB2	: UINT;				//ntHMI_Pir_SetValue i gammel kode
	uiSPLuxLevel_MB			AT %MB6 	: UINT;				//intHMI_Lux_SetValue i gammel kode
	uiBallastOnHours_MB		AT %MB14 	: UINT;				//dintHMILysbraendtimer1 i gammel kode
	byOnHoursOverflowCount				: BYTE;
END_VAR

A_Buttons();
A_LightCtrl();
A_ModbusComm();
A_Sensor();

ACTION A_Buttons:
bTopButtonZone1		:= GVL_EnOcean.strEnOceanSwitch_Gang_3_109_PladeA.bT1_ON OR bTopButtonZone1_Visu;
bBottomButtonZone1	:= GVL_EnOcean.strEnOceanSwitch_Gang_3_109_PladeA.bT1_OFF OR bBottomButtonZone1_Visu;
END_ACTION

ACTION A_LightCtrl:
bNeighborRoomsPir	:= 		 P_Gang_4_208.bPirActive_MB OR
 GVL_AHDataModbus.arrAH_NeighborRoomsPir  [4] [0] OR //2-1 
GVL_AHDataModbus.arrAH_NeighborRoomsPir  [4] [1] OR  //2-1 
GVL_AHDataModbus.arrAH_NeighborRoomsPir  [4] [2] OR //2-1 
GVL_AHDataModbus.arrAH_NeighborRoomsPir  [18] [0] OR//5-1
GVL_AHDataModbus.arrAH_NeighborRoomsPir  [18] [1]OR //5-1
GVL_AHDataModbus.arrAH_NeighborRoomsPir  [5] [0] OR //2-2
GVL_AHDataModbus.arrAH_NeighborRoomsPir  [5] [1] OR //2-2
GVL_AHDataModbus.arrAH_NeighborRoomsPir  [5] [2] OR //2-2
GVL_AHDataModbus.arrAH_NeighborRoomsPir  [5] [3] OR //2-2
GVL_AHDataModbus.arrAH_NeighborRoomsPir  [5] [4] OR //2-2
GVL_AHDataModbus.arrAH_NeighborRoomsPir  [5] [5] OR //2-2
GVL_AHDataModbus.arrAH_NeighborRoomsPir  [9] [0] OR //3-2 
GVL_AHDataModbus.arrAH_NeighborRoomsPir  [9] [1] OR //3-2 
GVL_AHDataModbus.arrAH_NeighborRoomsPir  [9] [2]  OR //3-2 
GVL_AHDataModbus.arrAH_NeighborRoomsPir  [14] [0] OR //4-2 
GVL_AHDataModbus.arrAH_NeighborRoomsPir [14] [1] OR //4-2 
GVL_AHDataModbus.arrAH_NeighborRoomsPir  [19] [0] OR //5-2 
GVL_AHDataModbus.arrAH_NeighborRoomsPir [19] [1] OR //5-2 
GVL_AHDataModbus.arrAH_NeighborRoomsPir [19] [2];  //5-2


//gruppe 5
arrfbLysGruppe[1]( 
	nZoneID:= 1, 
	bButtonZone1:= bTopButtonZone1,
	bBottomButtonZone1 := bBottomButtonZone1,
	//bTopButtonOverride := (GVL_EnOcean.strEnOceanSwitch_AtriumNiveau_PladeB.bT2_ON OR GVL_EnOcean.strEnOceanSwitch_AtriumNiveau_Service.bT2_ON),
	//bBottomButtonOverride := (GVL_EnOcean.strEnOceanSwitch_AtriumNiveau_PladeB.bT2_OFF OR GVL_EnOcean.strEnOceanSwitch_AtriumNiveau_Service.bT2_OFF),
	bButtonZone2:= bButtonZone2,
	bNeighborRoomsPir	:=	bNeighborRoomsPir,
	fLuxOn:= fLuxOn, 
	fLuxDim:= fLuxDim, 
	tPIRDim:= tPIRDim, 
	tPIROff:= tPIROff, 
	fOffsetSec:= fOffsetSec, 
	bReInit:= , 
	stDaliSetup:= arrstDaliSetupGruppe[1], 
	ipCommunication_Prim:= P_DALI_Background.arrfbKL6821Communication[arrDALI_LINE_NUM_LIGHT[1]], 
	ipCommunication_Sec:= P_DALI_Background.arrfbKL6821Communication[arrDALI_LINE_NUM_LIGHT[1]], //samme som lyslinjen, hvis den ikke eksisterer
	ipCommunication_Supl:= P_DALI_Background.arrfbKL6821Communication[arrDALI_LINE_NUM_LIGHT[1]],//samme som lyslinjen, hvis den ikke eksisterer 
	fMinOutputPowerLevelRoom:= 15, 
	fMaxOutputPowerLevelRoom:= 100, 
	nCycleTimeInMS:= SH_Light.DALI_Param.nPlcTaskCycleTimeInMS*nDimCmdCycleTimeFactor,  //Used only for dim. Factor=2 makes dimming smooth
	bRunTuning:= arrRunTuningGruppe[1], 
	bOccupiedRoom=> , 
	bError_Prim=> , 
	nError_Prim=> , 
	stTuneData:=arrstTuneDataGruppe[1] , 
	stPirSensorData:= stPirSensorData, 					//samme sensordata
	stLiveData:= arrstLiveDataGruppe[1]);

//gruppe 14	
arrfbLysGruppe[2]( 
	nZoneID:= 1, 
	bButtonZone1:= bTopButtonZone1,
	bBottomButtonZone1 := bBottomButtonZone1,
//	bTopButtonOverride := (GVL_EnOcean.strEnOceanSwitch_AtriumNiveau_PladeB.bT2_ON OR GVL_EnOcean.strEnOceanSwitch_AtriumNiveau_Service.bT2_ON),
//	bBottomButtonOverride := (GVL_EnOcean.strEnOceanSwitch_AtriumNiveau_PladeB.bT2_OFF OR GVL_EnOcean.strEnOceanSwitch_AtriumNiveau_Service.bT2_OFF),
	bButtonZone2:= bButtonZone2,
	bNeighborRoomsPir	:=	bNeighborRoomsPir,
	fLuxOn:= fLuxOn, 
	fLuxDim:= fLuxDim, 
	tPIRDim:= tPIRDim, 
	tPIROff:= tPIROff, 
	fOffsetSec:= fOffsetSec, 
	bReInit:= , 
	stDaliSetup:= arrstDaliSetupGruppe[2], 
	ipCommunication_Prim:= P_DALI_Background.arrfbKL6821Communication[arrDALI_LINE_NUM_LIGHT[2]], 
	ipCommunication_Sec:= P_DALI_Background.arrfbKL6821Communication[arrDALI_LINE_NUM_LIGHT[2]], //samme som lyslinjen, hvis den ikke eksisterer
	ipCommunication_Supl:= P_DALI_Background.arrfbKL6821Communication[arrDALI_LINE_NUM_LIGHT[2]], //samme som lyslinjen, hvis den ikke eksisterer 
	fMinOutputPowerLevelRoom:= 15, 
	fMaxOutputPowerLevelRoom:= 100, 
	nCycleTimeInMS:= SH_Light.DALI_Param.nPlcTaskCycleTimeInMS*nDimCmdCycleTimeFactor,  //Used only for dim. Factor=2 makes dimming smooth
	bRunTuning:= arrRunTuningGruppe[2], 
	bOccupiedRoom=> , 
	bError_Prim=> , 
	nError_Prim=> , 
	stTuneData:=arrstTuneDataGruppe[2] , 
	stPirSensorData:= stPirSensorData, 					//samme sensordata
	stLiveData:= arrstLiveDataGruppe[2]);
END_ACTION

ACTION A_ModbusComm:
//Manage data for modbus communication

//Manage data for read-only in PLC
stRoomDataPLC.bPirActive			:= stPirSensorData.bPrc;
stRoomDataPLC.uiActLuxLevel			:= TO_UINT(TRUNC(stPirSensorData.fBrightness));
stRoomDataPLC.uiActLightLevelPct	:= TO_UINT(TRUNC(arrfbLysGruppe[1].fbBallast.fActlLgtLvl_Prim));
		//stRoomDataPLC.uiActLightLevelPct	:= TO_UINT(TRUNC(fbLys.fbBallast.fActlLgtLvl_Prim)); //if only one group light control
stRoomDataPLC.uiBallastOnHours		:= uiBallastOnHours_MB; //The calculation for BallastOnHours is stored directly to the MB register below


//Assign data for read-only to MB registers
bPirActive_MB			:= stRoomDataPLC.bPirActive;
uiActLuxLevel_MB		:= stRoomDataPLC.uiActLuxLevel;
uiActLightLevelPct_MB	:= stRoomDataPLC.uiActLightLevelPct;

	//calculate BallastOnHours
	fbBallastOnHours(
		bEnableHourCount	:= bEnableHourCount,
		bPauseCount			:= arrfbLysGruppe[1].fbLightCtrl.bOffZone1,
		uiOnHours			:= uiBallastOnHours_MB,			//OnHours is updated here
		byOverflowCount		:= byOnHoursOverflowCount);


//Manage data for read/write for both PLC and MB registers
fbWriteSPLuxLevel(	nMaxValOut	:= uiMaxLuxLevel,
					nValIn1		:= uiSPLuxLevel_MB,		//nValIn1 takes priotity in case of download or restart
					nValIn2		:= stRoomDataPLC.uiSpLuxLevel,
					nValOut		=> uiLuxOn
				);


fbWritePirDelayTIme(	nMaxValOut	:= uiMaxPirOffMinutes,
						nValIn1		:= uiPirOffDelayTime_MB,		//nValIn1 takes priotity in case of download or restart
						nValIn2		:= stRoomDataPLC.uiPirOffDelayTime,
						nValOut		=> uiPirOffMinutes
					);
					

//Convert read/write modbus data to appropriate datatypes in PLC
fLuxOn	:= TO_REAL(uiLuxOn);			
tPIROff	:= TO_TIME(uiPirOffMinutes*udTimeScaling); //Time conversion defaults to ms

fLuxDim	:= TO_REAL(stRoomDataPLC.uiSpDimLuxLevel);			
tPIRDim	:= TO_TIME(stRoomDataPLC.uiPirDimDelayTime*udTimeScaling); //Time conversion defaults to ms
END_ACTION

ACTION A_Sensor:

fbSensor.ipCommunication := P_DALI_Background.arrfbKL6821Communication[Sensor_DALI_LINE_NUM];

(*//only 1 sensor
fbSensor(
	byShrtAdr:= bySensorAddr,
	bInitialize:= bInitialize, 
	DALI_LINE_NUM:= Sensor_DALI_LINE_NUM, 
 	//bCancelHoldTimerOccupancy:= bCancelHoldTimerOccupancy, 
	stSensorSetup := stDaliSensorSetup,
	bInitErr=> bInitErr, 
	bInitDone=> bInitDone,
	stPirSensorData:= stPirSensorData, 
	arrSensorScales:= arrSensorScales);
	*)

//several sensors	
fbSensor(
	arrShrtAdr:= arrSensorAddr,
	bInitialize:= bInitialize, 
	DALI_LINE_NUM:= Sensor_DALI_LINE_NUM, 
 	//bCancelHoldTimerOccupancy:= bCancelHoldTimerOccupancy, 
	stSensorSetup := stDaliSensorSetup,
	arrInitErr=> arrInitErr, 
	arrInitDone=> arrInitDone,
	stPirSensorData:= stPirSensorData, 
	arrSensorScales:= arrSensorScales);
END_ACTION

END_PROGRAM

// ---- POUs/Alle_Rum/Gange/Gang_4_208/P_Gang_4_208.TcPOU
PROGRAM P_Gang_4_208
VAR
(*Gangen består af to lysgrupper - L2G6 og L1G15
Begge grupper afhænger af samme PIR-input - pir-adr. 6, 7, 8, 9 og 10 - på DALI-linje 2.
Derfor oprettes to adskilte reguleringer med samme PV. Dvs., at knapfunktion og pirfunktion forbliver den samme.

En anden del af af hele gangen styres fra AH4_3. De to dele nabostyres med PIR-signaler over modbus-kommunikation*)
/////////////////////////////////
(*Gangen består af to lysgrupper - 4 og 4 - på to forskellige DALI-linjer - 2 og 1 henh..
Begge grupper afhænger af samme PIR-input - pir-adr. 6, 7, 8, 9 og 10 - på DALI-linje 2.
Derfor oprettes to adskilte reguleringer med samme PV. Dvs., at knapfunktion og pirfunktion forbliver den samme.

En anden del af af hele gangen styres fra AH4_3. De to dele nabostyres med PIR-signaler over modbus-kommunikation*)

	arrfbLysGruppe			: ARRAY [1..2] OF FB_Light_Type_B;
	arrstDaliSetupGruppe	: ARRAY[1..2] OF SH_Light.ST_DALI_RoomSetup := 
	
													[(	byShrtAdr_Prim := 25, 
														byGrpAdr_Prim := 5, 
														eMod_Prim := E_DALIAddressType.Group, 
														byShrtAdr_Sec := 1, 
														byGrpAdr_Sec := 1, 
														eMod_Sec := E_DALIAddressType.Short, 
														//byShrtAdr_Supl := 1,
														//eMod_Supl := E_DALIADDRESSTYPE.Group,
                                                        byGrpAdr_Supl := 1, 
														DALI_LINE_NUM_PRIM := arrDALI_LINE_NUM_LIGHT[1], 
														DALI_LINE_NUM_SEC := 0, //0 = ingen zonestyring/vinduerække
														DALI_LINE_NUM_SUPL := arrDALI_LINE_NUM_PENDANTS[1]),
														
													(	byShrtAdr_Prim := 20, 
														byGrpAdr_Prim := 5, 
														eMod_Prim := E_DALIAddressType.Group, 
														byShrtAdr_Sec := 1, 
														byGrpAdr_Sec := 1, 
														eMod_Sec := E_DALIAddressType.Short, 
														byShrtAdr_Supl := 1, 
														DALI_LINE_NUM_PRIM := arrDALI_LINE_NUM_LIGHT[2], 
														DALI_LINE_NUM_SEC := 0, 
														DALI_LINE_NUM_SUPL := arrDALI_LINE_NUM_PENDANTS[2])];
														
	arrstLiveDataGruppe		: ARRAY [1..2] OF SH_Light.ST_LiveData;
	//stLiveData AT %MB22	: SH_Light.ST_LiveData;
	
	arrRunTuningGruppe: ARRAY[1..2] OF BOOL;
	
	
	
	bTopButtonZone1			: BOOL;
	bTopButtonZone1_Visu	: BOOL;
	bBottomButtonZone1		: BOOL;
	bBottomButtonZone1_Visu	: BOOL;
	bButtonZone2			: BOOL;
	bNeighborRoomsPir		: BOOL;
	fLuxOn					: REAL; 
	fLuxDim					: REAL;
	tPIRDim					: TIME;
	tPIROff					: TIME;
	fOffsetSec				: REAL := 20;

//Digital In
//    bDigitalPir AT %I*      : BOOL ;    

// Sensor Settings
	//fbSensor					: SH_Light.FB_NIKO_P46xx_1Pcs;
	fbSensor					: SH_Light.FB_NIKO_P46xx_3Pcs;
	//bySensorAddr				: BYTE := 17;
	arrSensorAddr				: ARRAY[1..3] OF BYTE := [2,3,4];
	bInitialize					: BOOL := TRUE;
	stDaliSensorSetup			: ST_DALI_NIKOP46SetupData;
	//bInitErr					: BOOL;
	//bInitDone					: BOOL;
	arrInitErr					: ARRAY [1..3] OF BOOL;
	arrInitDone					: ARRAY [1..3] OF BOOL;
	arrSensorScales				: ARRAY [1..10] OF SH_Light.ST_DALI_SensorScaleMode := [	(fMeassureMaxSensor := rMeassure_Zone8, fReadMaxSensor := rRead_Zone8),
																							(fMeassureMaxSensor := rMeassure_Zone8, fReadMaxSensor := rRead_Zone8),	
                                                                                            (fMeassureMaxSensor := rMeassure_Zone8, fReadMaxSensor := rRead_Zone8),																				
																						7(())];
	bCancelHoldTimerOccupancy	: BOOL;
(*	eEventPriorityOccupancy		: E_DALIEventPriority := E_DALIEVENTPRIORITY.Middle;
	nHoldTimerOccupancy			: WORD := 5; // Value in s. 	
	nReportTimerOccupancy		: BYTE := 120; // Value in s, Preset manufacturer value
	nDeadtimeTimerOccupancy		: WORD := 100; // Value in ms, Predefined Value of DALI Standard
	bCancelHoldTimerOccupancy	: BOOL;
	nSensitivityOccupancy		: BYTE:= 3; //setting Sensivity (0..4) 0 (Off), 1 (Min), 2(Low), 3(High) and 4 (Max)

	bEnableLuxEvent				: BOOL;
	eEventPriorityBrightness	: E_DALIEventPriority := E_DALIEVENTPRIORITY.Middle;
	nDeadtimeTimerBrightness	: WORD := 1500; // Value in ms, Predefined Value of DALI Standard
	nHysteresisBrightness		: BYTE := 2; // Value in %
	nHysteresisMinBrightness	: BYTE := 10; // Absolute Value, depending on the manufacturer specific resolution
	nReportTimerBrightness		: BYTE := 120; // Value in s, Preset manufacturer value
*)


//ModbusComm setup
	
	fbWriteSPLuxLevel			: SH_Light.FB_TwoVal_SelectOne_RTrigChange;
	fbWritePirDelayTIme			: SH_Light.FB_TwoVal_SelectOne_RTrigChange;
	stRoomDataPLC				: SH_Light.ST_RoomDataPLC	:=	(	uiPirOffDelayTime	:= 30,
																	uiSpLuxLevel		:= 500,
																	uiPirDimDelayTime	:= 15,
																	uiSpDimLuxLevel		:= 200
																);
	fbBallastOnHours			: SH_Light.FB_CountOnHours;
	bEnableHourCount			: BOOL := TRUE;
	
	//Non-persistent modbus data
	bPirActive_MB			AT%MX60.0	: BOOL;				//bPirLys i gammel kode
	uiActLuxLevel_MB		AT%MB64	: UINT;				//intHMIAktueltLux i gammel kode
	uiActLightLevelPct_MB	AT%MB68	: UINT;				//intDALI_Gruppe1_Lysniveau i gammel kode
	
	//For Conversion
	uiPirOffMinutes						: UINT;
	udTimeScaling						: UDINT := 60000;
	uiLuxOn								: UINT;
	
	//max values checks
	uiMaxLuxLevel						: UINT := 1023;
	uiMaxPirOffMinutes					: UINT := 180;
	
END_VAR

VAR CONSTANT
	Sensor_DALI_LINE_NUM: BYTE := 3;
	arrDALI_LINE_NUM_LIGHT: ARRAY[1..2] OF BYTE := [2,1]; //korrekt rækkefølge nødvendig //rækkefølge og linje 
	arrDALI_LINE_NUM_PENDANTS: ARRAY[1..2] OF BYTE := [0,0]; //korrekt rækkefølge nødvendig. 0 = ingen pendler
END_VAR
VAR PERSISTENT
	stPirSensorData: SH_Light.ST_DALI_Sensor;
	arrstTuneDataGruppe: ARRAY [1..2] OF SH_Light.ST_TuneData_EX;

	uiPirOffDelayTime_MB	AT%MB62	    : UINT;				//intHMI_Pir_SetValue i gammel kode
	uiSPLuxLevel_MB		    AT%MB66     : UINT;				//intHMI_Lux_SetValue i gammel kode
	uiBallastOnHours_MB	    AT%MB70	    : UINT;				//dintHMILysbraendtimer1 i gammel kode
	byOnHoursOverflowCount			    : BYTE;
END_VAR

///////)

A_Buttons();
A_LightCtrl();
A_ModbusComm();
A_Sensor();

ACTION A_Buttons:
bTopButtonZone1		:= bTopButtonZone1_Visu;
bBottomButtonZone1	:= bBottomButtonZone1_Visu;
END_ACTION

ACTION A_LightCtrl:
bNeighborRoomsPir	:=    GVL_AHDataModbus.arrAH_NeighborRoomsPir  [4] [0] OR //2-1 
GVL_AHDataModbus.arrAH_NeighborRoomsPir  [4] [1] OR  //2-1 
GVL_AHDataModbus.arrAH_NeighborRoomsPir  [4] [2] OR //2-1 
GVL_AHDataModbus.arrAH_NeighborRoomsPir  [18] [0] OR//5-1
GVL_AHDataModbus.arrAH_NeighborRoomsPir  [18] [1]OR //5-1
GVL_AHDataModbus.arrAH_NeighborRoomsPir  [5] [0] OR //2-2
GVL_AHDataModbus.arrAH_NeighborRoomsPir  [5] [1] OR //2-2
GVL_AHDataModbus.arrAH_NeighborRoomsPir  [5] [2] OR //2-2
GVL_AHDataModbus.arrAH_NeighborRoomsPir  [5] [3] OR //2-2
GVL_AHDataModbus.arrAH_NeighborRoomsPir  [5] [4] OR //2-2
GVL_AHDataModbus.arrAH_NeighborRoomsPir  [5] [5] OR //2-2
GVL_AHDataModbus.arrAH_NeighborRoomsPir  [9] [0] OR //3-2 
GVL_AHDataModbus.arrAH_NeighborRoomsPir  [9] [1] OR //3-2 
GVL_AHDataModbus.arrAH_NeighborRoomsPir  [9] [2]  OR //3-2 
GVL_AHDataModbus.arrAH_NeighborRoomsPir  [14] [0] OR //4-2 
GVL_AHDataModbus.arrAH_NeighborRoomsPir [14] [1] OR //4-2 
GVL_AHDataModbus.arrAH_NeighborRoomsPir  [19] [0] OR //5-2 
GVL_AHDataModbus.arrAH_NeighborRoomsPir [19] [1] OR //5-2 
GVL_AHDataModbus.arrAH_NeighborRoomsPir [19] [2];  //5-2

                       ;
//gruppe 6
arrfbLysGruppe[1]( 
	nZoneID:= 1, 
	bButtonZone1:= bTopButtonZone1,
	bBottomButtonZone1 := bBottomButtonZone1,
	bTopButtonOverride := (GVL_EnOcean.strEnOceanSwitch_AtriumNiveau_PladeB.bT2_ON OR GVL_EnOcean.strEnOceanSwitch_AtriumNiveau_Service.bT2_ON),
	bBottomButtonOverride := (GVL_EnOcean.strEnOceanSwitch_AtriumNiveau_PladeB.bT2_OFF OR GVL_EnOcean.strEnOceanSwitch_AtriumNiveau_Service.bT2_OFF),
	bButtonZone2:= bButtonZone2,
	bNoButtons := TRUE,
	bNeighborRoomsPir	:=	bNeighborRoomsPir,
	fLuxOn:= fLuxOn, 
	fLuxDim:= fLuxDim, 
	tPIRDim:= tPIRDim, 
	tPIROff:= tPIROff, 
	fOffsetSec:= fOffsetSec, 
	bReInit:= , 
	stDaliSetup:= arrstDaliSetupGruppe[1], 
	ipCommunication_Prim:= P_DALI_Background.arrfbKL6821Communication[arrDALI_LINE_NUM_LIGHT[1]], 
	ipCommunication_Sec:= P_DALI_Background.arrfbKL6821Communication[arrDALI_LINE_NUM_LIGHT[1]], //samme som lyslinjen, hvis den ikke eksisterer
	ipCommunication_Supl:= P_DALI_Background.arrfbKL6821Communication[arrDALI_LINE_NUM_LIGHT[1]],//samme som lyslinjen, hvis den ikke eksisterer 
	fMinOutputPowerLevelRoom:= 15, 
	fMaxOutputPowerLevelRoom:= 100, 
	nCycleTimeInMS:= SH_Light.DALI_Param.nPlcTaskCycleTimeInMS*nDimCmdCycleTimeFactor,  //Used only for dim. Factor=2 makes dimming smooth
	bRunTuning:= arrRunTuningGruppe[1], 
	bOccupiedRoom=> , 
	bError_Prim=> , 
	nError_Prim=> , 
	stTuneData:=arrstTuneDataGruppe[1] , 
	stPirSensorData:= stPirSensorData, 					//samme sensordata
	stLiveData:= arrstLiveDataGruppe[1]);

//gruppe 15	
arrfbLysGruppe[2]( 
	nZoneID:= 1, 
	bButtonZone1:= bTopButtonZone1,
	bBottomButtonZone1 := bBottomButtonZone1,
	bTopButtonOverride := (GVL_EnOcean.strEnOceanSwitch_AtriumNiveau_PladeB.bT2_ON OR GVL_EnOcean.strEnOceanSwitch_AtriumNiveau_Service.bT2_ON),
	bBottomButtonOverride := (GVL_EnOcean.strEnOceanSwitch_AtriumNiveau_PladeB.bT2_OFF OR GVL_EnOcean.strEnOceanSwitch_AtriumNiveau_Service.bT2_OFF),
	bButtonZone2:= bButtonZone2,
	bNoButtons := TRUE,
	bNeighborRoomsPir	:=	bNeighborRoomsPir,
	fLuxOn:= fLuxOn, 
	fLuxDim:= fLuxDim, 
	tPIRDim:= tPIRDim, 
	tPIROff:= tPIROff, 
	fOffsetSec:= fOffsetSec, 
	bReInit:= , 
	stDaliSetup:= arrstDaliSetupGruppe[2], 
	ipCommunication_Prim:= P_DALI_Background.arrfbKL6821Communication[arrDALI_LINE_NUM_LIGHT[2]], 
	ipCommunication_Sec:= P_DALI_Background.arrfbKL6821Communication[arrDALI_LINE_NUM_LIGHT[2]], //samme som lyslinjen, hvis den ikke eksisterer
	ipCommunication_Supl:= P_DALI_Background.arrfbKL6821Communication[arrDALI_LINE_NUM_LIGHT[2]], //samme som lyslinjen, hvis den ikke eksisterer 
	fMinOutputPowerLevelRoom:= 15, 
	fMaxOutputPowerLevelRoom:= 100, 
	nCycleTimeInMS:= SH_Light.DALI_Param.nPlcTaskCycleTimeInMS*nDimCmdCycleTimeFactor,  //Used only for dim. Factor=2 makes dimming smooth
	bRunTuning:= arrRunTuningGruppe[2], 
	bOccupiedRoom=> , 
	bError_Prim=> , 
	nError_Prim=> , 
	stTuneData:=arrstTuneDataGruppe[2] , 
	stPirSensorData:= stPirSensorData, 					//samme sensordata
	stLiveData:= arrstLiveDataGruppe[2]);
END_ACTION

ACTION A_ModbusComm:
//Manage data for modbus communication

//Manage data for read-only in PLC
stRoomDataPLC.bPirActive			:= stPirSensorData.bPrc;
stRoomDataPLC.uiActLuxLevel			:= TO_UINT(TRUNC(stPirSensorData.fBrightness));
stRoomDataPLC.uiActLightLevelPct	:= TO_UINT(TRUNC(arrfbLysGruppe[1].fbBallast.fActlLgtLvl_Prim));
		//stRoomDataPLC.uiActLightLevelPct	:= TO_UINT(TRUNC(fbLys.fbBallast.fActlLgtLvl_Prim)); //if only one group light control
stRoomDataPLC.uiBallastOnHours		:= uiBallastOnHours_MB; //The calculation for BallastOnHours is stored directly to the MB register below


//Assign data for read-only to MB registers
bPirActive_MB		:= stRoomDataPLC.bPirActive;
uiActLuxLevel_MB	:= stRoomDataPLC.uiActLuxLevel;

	//calculate BallastOnHours
	fbBallastOnHours(
		bEnableHourCount	:= bEnableHourCount,
		bPauseCount			:= arrfbLysGruppe[1].fbLightCtrl.bOffZone1,
		uiOnHours			:= uiBallastOnHours_MB,			//OnHours is updated here
		byOverflowCount		:= byOnHoursOverflowCount);


//Manage data for read/write for both PLC and MB registers
fbWriteSPLuxLevel(	nMaxValOut	:= uiMaxLuxLevel,
					nValIn1		:= uiSPLuxLevel_MB,		//nValIn1 takes priotity in case of download or restart
					nValIn2		:= stRoomDataPLC.uiSpLuxLevel,
					nValOut		=> uiLuxOn
				);


fbWritePirDelayTIme(	nMaxValOut	:= uiMaxPirOffMinutes,
						nValIn1		:= uiPirOffDelayTime_MB,		//nValIn1 takes priotity in case of download or restart
						nValIn2		:= stRoomDataPLC.uiPirOffDelayTime,
						nValOut		=> uiPirOffMinutes
					);
					

//Convert read/write modbus data to appropriate datatypes in PLC
fLuxOn	:= TO_REAL(uiLuxOn);			
tPIROff	:= TO_TIME(uiPirOffMinutes*udTimeScaling); //Time conversion defaults to ms

fLuxDim	:= TO_REAL(stRoomDataPLC.uiSpDimLuxLevel);			
tPIRDim	:= TO_TIME(stRoomDataPLC.uiPirDimDelayTime*udTimeScaling); //Time conversion defaults to ms
END_ACTION

ACTION A_Sensor:

fbSensor.ipCommunication := P_DALI_Background.arrfbKL6821Communication[Sensor_DALI_LINE_NUM];

(*//only 1 sensor
fbSensor(
	byShrtAdr:= bySensorAddr,
	bInitialize:= bInitialize, 
	DALI_LINE_NUM:= Sensor_DALI_LINE_NUM, 
 	//bCancelHoldTimerOccupancy:= bCancelHoldTimerOccupancy, 
	stSensorSetup := stDaliSensorSetup,
	bInitErr=> bInitErr, 
	bInitDone=> bInitDone,
	stPirSensorData:= stPirSensorData, 
	arrSensorScales:= arrSensorScales);
	*)

//several sensors	
fbSensor(
	arrShrtAdr:= arrSensorAddr,
	bInitialize:= bInitialize, 
	DALI_LINE_NUM:= Sensor_DALI_LINE_NUM, 
 	//bCancelHoldTimerOccupancy:= bCancelHoldTimerOccupancy, 
	stSensorSetup := stDaliSensorSetup,
	arrInitErr=> arrInitErr, 
	arrInitDone=> arrInitDone,
	stPirSensorData:= stPirSensorData, 
	arrSensorScales:= arrSensorScales);
END_ACTION

END_PROGRAM

// ---- POUs/Alle_Rum/Rum_Med_DALI_Pir/Rum_4_206/P_Rum_4_206.TcPOU
PROGRAM P_Rum_4_206
VAR
(*Rummet består af to lysgrupper - L1G1 og L2G1 - på to forskellige linjer
Begge grupper afhænger af samme PIR-input - pir-adr. 1 og 2 - på DALI-linje 1.
Derfor oprettes to adskilte reguleringer med samme PV. Dvs., at knapfunktion og pirfunktion forbliver den samme.
*)

	arrfbLysGruppe			: ARRAY [1..2] OF SH_Light.FB_Light_Type_A;
	arrstDaliSetupGruppe	: ARRAY [1..2] OF SH_Light.ST_DALI_RoomSetup := 
	
													[(	byShrtAdr_Prim := 1, 
														byGrpAdr_Prim := 1, 
														eMod_Prim := E_DALIAddressType.Group, 
														//byShrtAdr_Sec := 1, 
														//byGrpAdr_Sec := 1, 
														//eMod_Sec := E_DALIAddressType.Short, 
														//byShrtAdr_Supl := 1,
														//byGrpAdr_Supl := 1,
														//eMod_Supl := E_DALIADDRESSTYPE.Group,
														DALI_LINE_NUM_PRIM := arrDALI_LINE_NUM_LIGHT[1], 
														DALI_LINE_NUM_SEC := 0, //0 = ingen zonestyring/vinduerække
														DALI_LINE_NUM_SUPL := arrDALI_LINE_NUM_PENDANTS[1]),
														
													(	byShrtAdr_Prim := 4, 
														byGrpAdr_Prim := 1, 
														eMod_Prim := E_DALIAddressType.Group,
														//byShrtAdr_Sec := 1, 
														//byGrpAdr_Sec := 1, 
														//eMod_Sec := E_DALIAddressType.Short, 
														//byShrtAdr_Supl := 1,
														//byGrpAdr_Supl := 1,
														//eMod_Supl := E_DALIAddressType.Group, 
														DALI_LINE_NUM_PRIM := arrDALI_LINE_NUM_LIGHT[2], 
														DALI_LINE_NUM_SEC := 0, 
														DALI_LINE_NUM_SUPL := arrDALI_LINE_NUM_PENDANTS[2])];
														
	arrstLiveDataGruppe		: ARRAY [1..2] OF SH_Light.ST_LiveData;
	
	arrRunTuningGruppe: ARRAY[1..2] OF BOOL;
	
	bTopButtonZone1				: BOOL;
	bTopButtonZone1_Visu		: BOOL;
	bBottomButtonZone1			: BOOL;
	bBottomButtonZone1_Visu	: BOOL;
	bButtonZone2					: BOOL;
	bNeighborRoomsPir			: BOOL;
	fLuxOn								: REAL; 
	fLuxDim							: REAL;
	tPIRDim							: TIME;
	tPIROff							: TIME;
	fOffsetSec						: REAL := 20;
 

// Sensor Settings
	//fbSensor					: SH_Light.FB_NIKO_P46xx_1Pcs;
	fbSensor						: SH_Light.FB_NIKO_P46xx_2Pcs;
	//bySensorAddr				: BYTE := 17;
	arrSensorAddr				: ARRAY[1..2] OF BYTE := [1,2];
	bInitialize						: BOOL := TRUE;
	stDaliSensorSetup			: ST_DALI_NIKOP46SetupData;
	//bInitErr							: BOOL;
	//bInitDone						: BOOL;
	arrInitErr						: ARRAY [1..2] OF BOOL;
	arrInitDone					: ARRAY [1..2] OF BOOL;
	arrSensorScales				: ARRAY [1..10] OF SH_Light.ST_DALI_SensorScaleMode :=
																					[	(fMeassureMaxSensor := rMeassure_Zone5, fReadMaxSensor := rRead_Zone5),
																						(fMeassureMaxSensor := rMeassure_Zone5, fReadMaxSensor := rRead_Zone5),																			
																						8(())];
																																			
	bCancelHoldTimerOccupancy	: BOOL;
(*	eEventPriorityOccupancy		: E_DALIEventPriority := E_DALIEVENTPRIORITY.Middle;
	nHoldTimerOccupancy			: WORD := 5; // Value in s. 	
	nReportTimerOccupancy		: BYTE := 120; // Value in s, Preset manufacturer value
	nDeadtimeTimerOccupancy		: WORD := 100; // Value in ms, Predefined Value of DALI Standard
	bCancelHoldTimerOccupancy	: BOOL;
	nSensitivityOccupancy		: BYTE:= 3; //setting Sensivity (0..4) 0 (Off), 1 (Min), 2(Low), 3(High) and 4 (Max)

	bEnableLuxEvent				: BOOL;
	eEventPriorityBrightness	: E_DALIEventPriority := E_DALIEVENTPRIORITY.Middle;
	nDeadtimeTimerBrightness	: WORD := 1500; // Value in ms, Predefined Value of DALI Standard
	nHysteresisBrightness		: BYTE := 2; // Value in %
	nHysteresisMinBrightness	: BYTE := 10; // Absolute Value, depending on the manufacturer specific resolution
	nReportTimerBrightness		: BYTE := 120; // Value in s, Preset manufacturer value
*)


//ModbusComm setup
	
	fbWriteSPLuxLevel				: SH_Light.FB_TwoVal_SelectOne_RTrigChange;
	fbWritePirDelayTIme			: SH_Light.FB_TwoVal_SelectOne_RTrigChange;
	stRoomDataPLC					: SH_Light.ST_RoomDataPLC	:=	(	uiPirOffDelayTime	:= 30,
																										uiSpLuxLevel			:= 500,
																										uiPirDimDelayTime	:= 15,
																										uiSpDimLuxLevel		:= 200);
																
	fbBallastOnHours					: SH_Light.FB_CountOnHours;
	bEnableHourCount				: BOOL := TRUE;
	
	//Non-persistent modbus data
	bPirActive_MB					AT%MX22.0	: BOOL;				//bPirLys i gammel kode
	uiActLuxLevel_MB			AT%MB26		: UINT;				//intHMIAktueltLux i gammel kode
	uiActLightLevelPct_MB	AT%MB32		: UINT;				//intDALI_Gruppe1_Lysniveau i gammel kode
	
	//For Conversion
	uiPirOffMinutes						: UINT;
	udTimeScaling						: UDINT := 60000;
	uiLuxOn								: UINT;
	
	//max values checks
	uiMaxLuxLevel						: UINT := 1023;
	uiMaxPirOffMinutes					: UINT := 180;
	
END_VAR

VAR CONSTANT
	Sensor_DALI_LINE_NUM					: BYTE := 1;
	arrDALI_LINE_NUM_LIGHT				: ARRAY[1..2] OF BYTE := [1,2]; //korrekt rækkefølge nødvendig //rækkefølge og linje 
	arrDALI_LINE_NUM_PENDANTS	: ARRAY[1..2] OF BYTE := [0,0]; //korrekt rækkefølge nødvendig. 0 = ingen pendler
END_VAR

VAR PERSISTENT
	stPirSensorData										: SH_Light.ST_DALI_Sensor;
	arrstTuneDataGruppe								: ARRAY [1..2] OF SH_Light.ST_TuneData_EX;

	uiPirOffDelayTime_MB		AT%MB24	    : UINT;				//intHMI_Pir_SetValue i gammel kode
	uiSPLuxLevel_MB		    AT%MB28    	: UINT;				//intHMI_Lux_SetValue i gammel kode
	uiBallastOnHours_MB	    AT%MB36	    : UINT;				//dintHMILysbraendtimer1 i gammel kode
	byOnHoursOverflowCount			   				: BYTE;
END_VAR

A_Buttons();
A_LightCtrl();
A_ModbusComm();
A_Sensor();

ACTION A_Buttons:
bTopButtonZone1		:= GVL_EnOcean.strEnOceanSwitch_Rum_4_206_Indgang.bT1_ON OR
									GVL_EnOcean.strEnOceanSwitch_Rum_4_206_Ekstra.bT2_ON OR
									bTopButtonZone1_Visu;
bBottomButtonZone1	:= GVL_EnOcean.strEnOceanSwitch_Rum_4_206_Indgang.bT1_OFF OR
									GVL_EnOcean.strEnOceanSwitch_Rum_4_206_Ekstra.bT2_OFF OR
									bBottomButtonZone1_Visu;
END_ACTION

ACTION A_LightCtrl:
                       ;
//gruppe L1G1
arrfbLysGruppe[1]( 
	nZoneID:= 1, 
	bButtonZone1:= bTopButtonZone1,
	bBottomButtonZone1 := bBottomButtonZone1,
	//bButtonZone2:= bButtonZone2,
	fLuxOn:= fLuxOn, 
	fLuxDim:= fLuxDim, 
	tPIRDim:= tPIRDim, 
	tPIROff:= tPIROff, 
	fOffsetSec:= fOffsetSec, 
	bReInit:= , 
	stDaliSetup:= arrstDaliSetupGruppe[1], 
	ipCommunication_Prim:= P_DALI_Background.arrfbKL6821Communication[arrDALI_LINE_NUM_LIGHT[1]], 
	//ipCommunication_Sec:= P_DALI_Background.arrfbKL6821Communication[arrDALI_LINE_NUM_LIGHT[1]],
	//ipCommunication_Supl:= P_DALI_Background.arrfbKL6821Communication[arrDALI_LINE_NUM_PENDANTS[1]], 
	fMinOutputPowerLevelRoom:= 15, 
	fMaxOutputPowerLevelRoom:= 100, 
	nCycleTimeInMS:= SH_Light.DALI_Param.nPlcTaskCycleTimeInMS*nDimCmdCycleTimeFactor,  //Used only for dim. Factor=2 makes dimming smooth
	bRunTuning:= arrRunTuningGruppe[1], 
	bOccupiedRoom=> , 
	bError_Prim=> , 
	nError_Prim=> , 
	stTuneData:=arrstTuneDataGruppe[1] , 
	stPirSensorData:= stPirSensorData, 					//samme sensordata
	stLiveData:= arrstLiveDataGruppe[1]);

//gruppe 15	
arrfbLysGruppe[2]( 
	nZoneID:= 1, 
	bButtonZone1:= bTopButtonZone1,
	bBottomButtonZone1 := bBottomButtonZone1,
	//bButtonZone2:= bButtonZone2,
	fLuxOn:= fLuxOn, 
	fLuxDim:= fLuxDim, 
	tPIRDim:= tPIRDim, 
	tPIROff:= tPIROff, 
	fOffsetSec:= fOffsetSec, 
	bReInit:= , 
	stDaliSetup:= arrstDaliSetupGruppe[2], 
	ipCommunication_Prim:= P_DALI_Background.arrfbKL6821Communication[arrDALI_LINE_NUM_LIGHT[2]], 
	//ipCommunication_Sec:= P_DALI_Background.arrfbKL6821Communication[arrDALI_LINE_NUM_LIGHT[2]],
	//ipCommunication_Supl:= P_DALI_Background.arrfbKL6821Communication[arrDALI_LINE_NUM_PENDANTS[2]], 
	fMinOutputPowerLevelRoom:= 15, 
	fMaxOutputPowerLevelRoom:= 100, 
	nCycleTimeInMS:= SH_Light.DALI_Param.nPlcTaskCycleTimeInMS*nDimCmdCycleTimeFactor,  //Used only for dim. Factor=2 makes dimming smooth
	bRunTuning:= arrRunTuningGruppe[2], 
	bOccupiedRoom=> , 
	bError_Prim=> , 
	nError_Prim=> , 
	stTuneData:=arrstTuneDataGruppe[2] , 
	stPirSensorData:= stPirSensorData, 					//samme sensordata
	stLiveData:= arrstLiveDataGruppe[2]);
END_ACTION

ACTION A_ModbusComm:
//Manage data for modbus communication

//Manage data for read-only in PLC
stRoomDataPLC.bPirActive			:= stPirSensorData.bPrc;
stRoomDataPLC.uiActLuxLevel			:= TO_UINT(TRUNC(stPirSensorData.fBrightness));
stRoomDataPLC.uiActLightLevelPct	:= TO_UINT(TRUNC(arrfbLysGruppe[1].fbBallast.fActlLgtLvl_Prim));
		//stRoomDataPLC.uiActLightLevelPct	:= TO_UINT(TRUNC(fbLys.fbBallast.fActlLgtLvl_Prim)); //if only one group light control
stRoomDataPLC.uiBallastOnHours		:= uiBallastOnHours_MB; //The calculation for BallastOnHours is stored directly to the MB register below


//Assign data for read-only to MB registers
bPirActive_MB		:= stRoomDataPLC.bPirActive;
uiActLuxLevel_MB	:= stRoomDataPLC.uiActLuxLevel;

	//calculate BallastOnHours
	fbBallastOnHours(
		bEnableHourCount	:= bEnableHourCount,
		bPauseCount			:= arrfbLysGruppe[1].fbLightCtrl.bOffZone1,
		uiOnHours			:= uiBallastOnHours_MB,			//OnHours is updated here
		byOverflowCount		:= byOnHoursOverflowCount);


//Manage data for read/write for both PLC and MB registers
fbWriteSPLuxLevel(	nMaxValOut	:= uiMaxLuxLevel,
					nValIn1		:= uiSPLuxLevel_MB,		//nValIn1 takes priotity in case of download or restart
					nValIn2		:= stRoomDataPLC.uiSpLuxLevel,
					nValOut		=> uiLuxOn
				);


fbWritePirDelayTIme(	nMaxValOut	:= uiMaxPirOffMinutes,
						nValIn1		:= uiPirOffDelayTime_MB,		//nValIn1 takes priotity in case of download or restart
						nValIn2		:= stRoomDataPLC.uiPirOffDelayTime,
						nValOut		=> uiPirOffMinutes
					);
					

//Convert read/write modbus data to appropriate datatypes in PLC
fLuxOn	:= TO_REAL(uiLuxOn);			
tPIROff	:= TO_TIME(uiPirOffMinutes*udTimeScaling); //Time conversion defaults to ms

fLuxDim	:= TO_REAL(stRoomDataPLC.uiSpDimLuxLevel);			
tPIRDim	:= TO_TIME(stRoomDataPLC.uiPirDimDelayTime*udTimeScaling); //Time conversion defaults to ms
END_ACTION

ACTION A_Sensor:

fbSensor.ipCommunication := P_DALI_Background.arrfbKL6821Communication[Sensor_DALI_LINE_NUM];

(*//only 1 sensor
fbSensor(
	byShrtAdr:= bySensorAddr,
	bInitialize:= bInitialize, 
	DALI_LINE_NUM:= Sensor_DALI_LINE_NUM, 
 	//bCancelHoldTimerOccupancy:= bCancelHoldTimerOccupancy, 
	stSensorSetup := stDaliSensorSetup,
	bInitErr=> bInitErr, 
	bInitDone=> bInitDone,
	stPirSensorData:= stPirSensorData, 
	arrSensorScales:= arrSensorScales);
	*)

//several sensors	
fbSensor(
	arrShrtAdr:= arrSensorAddr,
	bInitialize:= bInitialize, 
	DALI_LINE_NUM:= Sensor_DALI_LINE_NUM, 
 	//bCancelHoldTimerOccupancy:= bCancelHoldTimerOccupancy, 
	stSensorSetup := stDaliSensorSetup,
	arrInitErr=> arrInitErr, 
	arrInitDone=> arrInitDone,
	stPirSensorData:= stPirSensorData, 
	arrSensorScales:= arrSensorScales);
END_ACTION

END_PROGRAM

// ---- POUs/Alle_Rum/Rum_Med_DALI_Pir/Rum_4_207/P_Rum_4_207.TcPOU
PROGRAM P_Rum_4_207
VAR
//Light

	fbLys			: FB_Light_Type_A;
	
	stDaliSetup	: SH_Light.ST_DALI_RoomSetup := (
														byShrtAdr_Prim	:= 10, 
														byGrpAdr_Prim		:= 2, 
														eMod_Prim			:= E_DALIAddressType.Group, 
														//byShrtAdr_Sec	:= 1, 
														//byGrpAdr_Sec	:= 1, 
														//eMod_Sec			:= E_DALIAddressType.Short, 
														//byShrtAdr_Supl		:= 1,
														//byGrpAdr_Supl		:= 1,
														//eMod_Supl			:= Tc3_DALI.E_DALIAddressType.Short, 
														DALI_LINE_NUM_PRIM := DALI_LINE_NUM_LIGHT, 
														DALI_LINE_NUM_SEC := 0, 
														DALI_LINE_NUM_SUPL := DALI_LINE_NUM_PENDANT);
														
	stLiveData					: SH_Light.ST_LiveData;
	bRunTuning					: BOOL;
	
	bTopButtonZone1			: BOOL;
	bTopButtonZone1_Visu	: BOOL;
	bBottomButtonZone1		: BOOL;
	bBottomButtonZone1_Visu	: BOOL;
	bButtonZone2				: BOOL;
	fLuxOn							: REAL;
	fLuxDim						: REAL;
	tPIRDim						: TIME;
	tPIROff						: TIME;
	fOffsetSec					: REAL := 20;
	bOccupiedRoom			: BOOL;
	
// Sensor Settings
	fbSensor						: SH_Light.FB_NIKO_P46xx_1Pcs;
	//fbSensor						: SH_Light.FB_NIKO_P46xx_2Pcs;
	bySensorAddr				: BYTE := 1;
	//arrSensorAddr				: ARRAY[1..2] OF BYTE := [3,4];
	bInitialize						: BOOL := TRUE;
	stDaliSensorSetup			: ST_DALI_NIKOP46SetupData;
	bInitErr							: BOOL;
	bInitDone						: BOOL;
	//arrInitErr						: ARRAY [1..2] OF BOOL;
	//arrInitDone					: ARRAY [1..2] OF BOOL;
	arrSensorScales				: ARRAY [1..10] OF SH_Light.ST_DALI_SensorScaleMode :=
																						[	(fMeassureMaxSensor := rMeassure_Zone5, fReadMaxSensor := rRead_Zone5),
																							9(())];
	bCancelHoldTimerOccupancy	: BOOL;
(*	eEventPriorityOccupancy		: E_DALIEventPriority := E_DALIEVENTPRIORITY.Middle;
	nHoldTimerOccupancy			: WORD := 5; // Value in s. 	
	nReportTimerOccupancy		: BYTE := 120; // Value in s, Preset manufacturer value
	nDeadtimeTimerOccupancy		: WORD := 100; // Value in ms, Predefined Value of DALI Standard
	bCancelHoldTimerOccupancy	: BOOL;
	nSensitivityOccupancy		: BYTE:= 3; //setting Sensivity (0..4) 0 (Off), 1 (Min), 2(Low), 3(High) and 4 (Max)

	bEnableLuxEvent				: BOOL;
	eEventPriorityBrightness	: E_DALIEventPriority := E_DALIEVENTPRIORITY.Middle;
	nDeadtimeTimerBrightness	: WORD := 1500; // Value in ms, Predefined Value of DALI Standard
	nHysteresisBrightness		: BYTE := 2; // Value in %
	nHysteresisMinBrightness	: BYTE := 10; // Absolute Value, depending on the manufacturer specific resolution
	nReportTimerBrightness		: BYTE := 120; // Value in s, Preset manufacturer value
*)

//ModbusComm setup
	
	fbWriteSPLuxLevel				: SH_Light.FB_TwoVal_SelectOne_RTrigChange;
	fbWritePirDelayTIme			: SH_Light.FB_TwoVal_SelectOne_RTrigChange;
	stRoomDataPLC					: SH_Light.ST_RoomDataPLC	:=	(	uiPirOffDelayTime	:= 30,
																										uiSpLuxLevel			:= 500,
																										uiPirDimDelayTime	:= 15,
																										uiSpDimLuxLevel		:= 200);
																
	fbBallastOnHours					: SH_Light.FB_CountOnHours;
	bEnableHourCount				: BOOL := TRUE;
	
	//Non-persistent modbus data
	bPirActive_MB					AT%MX44.0	: BOOL;				//bPirLys i gammel kode
	uiActLuxLevel_MB			AT%MB48		: UINT;				//intHMIAktueltLux i gammel kode
	uiActLightLevelPct_MB	AT%MB52		: UINT;				//intDALI_Gruppe1_Lysniveau i gammel kode
	
	//For Conversion
	uiPirOffMinutes						: UINT;
	udTimeScaling						: UDINT := 60000;
	uiLuxOn								: UINT;
	
	//max values checks
	uiMaxLuxLevel						: UINT := 1023;
	uiMaxPirOffMinutes				: UINT := 180;

END_VAR

VAR CONSTANT
	Sensor_DALI_LINE_NUM: BYTE := 3;
	DALI_LINE_NUM_LIGHT: BYTE := 1;
	DALI_LINE_NUM_PENDANT: BYTE :=0;
END_VAR
VAR PERSISTENT
	stPirSensorData: SH_Light.ST_DALI_Sensor;
	stTuneData: SH_Light.ST_TuneData_EX;
	
	uiPirOffDelayTime_MB		AT%MB46	    : UINT;				//intHMI_Pir_SetValue i gammel kode
	uiSPLuxLevel_MB		    AT%MB50    	: UINT;				//intHMI_Lux_SetValue i gammel kode
	uiBallastOnHours_MB	    AT%MB54	    : UINT;				//dintHMILysbraendtimer1 i gammel kode
	byOnHoursOverflowCount			   				: BYTE;
END_VAR

A_Buttons();
A_LightCtrl();
A_ModbusComm();
A_Sensor();

ACTION A_Buttons:
bTopButtonZone1		:= GVL_EnOcean.strEnOceanSwitch_Rum_4_207_Indgang.bT2_ON OR
									GVL_EnOcean.strEnOceanSwitch_Rum_4_207_Ekstra.bT1_ON OR
									bTopButtonZone1_Visu;
bBottomButtonZone1	:= GVL_EnOcean.strEnOceanSwitch_Rum_4_207_Indgang.bT2_OFF OR
									GVL_EnOcean.strEnOceanSwitch_Rum_4_207_Ekstra.bT1_OFF OR
									bBottomButtonZone1_Visu;
END_ACTION

ACTION A_LightCtrl:

fbLys(
	nZoneID:= 1, 
	bButtonZone1:= bTopButtonZone1,
	bBottomButtonZone1 := bBottomButtonZone1, 
	//bButtonZone2:= bButtonZone2, 
	fLuxOn:= fLuxOn, 
	fLuxDim:= fLuxDim, 
	tPIRDim:= tPIRDim, 
	tPIROff:= tPIROff, 
	fOffsetSec:= fOffsetSec, 
	bReInit:= , 
	stDaliSetup:= stDaliSetup, 
	ipCommunication_Prim:= P_DALI_Background.arrfbKL6821Communication[DALI_LINE_NUM_LIGHT], 
	//ipCommunication_Sec:= P_DALI_Background.arrfbKL6821Communication[DALI_LINE_NUM_LIGHT], 
	//ipCommunication_Supl:= P_DALI_Background.arrfbKL6821Communication[DALI_LINE_NUM_PENDANT],
	fMinOutputPowerLevelRoom:= 15, 
	fMaxOutputPowerLevelRoom:= 100, 
	nCycleTimeInMS:= SH_Light.DALI_Param.nPlcTaskCycleTimeInMS*nDimCmdCycleTimeFactor,  //Used only for dim. Factor=2 makes dimming smooth
	bRunTuning:= bRunTuning, 
	bOccupiedRoom=> bOccupiedRoom, 
	bError_Prim=> , 
	nError_Prim=> , 
	stTuneData:=stTuneData , 
	stPirSensorData:= stPirSensorData, 
	stLiveData:= stLiveData);
END_ACTION

ACTION A_ModbusComm:
//Manage data for modbus communication

//Manage data for read-only in PLC
stRoomDataPLC.bPirActive			:= stPirSensorData.bPrc;
stRoomDataPLC.uiActLuxLevel			:= TO_UINT(TRUNC(stPirSensorData.fBrightness));
stRoomDataPLC.uiActLightLevelPct	:= TO_UINT(TRUNC(fblys.fbBallast.fActlLgtLvl_Prim));
		//stRoomDataPLC.uiActLightLevelPct	:= TO_UINT(TRUNC(fbLys.fbBallast.fActlLgtLvl_Prim)); //if only one group light control
stRoomDataPLC.uiBallastOnHours		:= uiBallastOnHours_MB; //The calculation for BallastOnHours is stored directly to the MB register below


//Assign data for read-only to MB registers
bPirActive_MB		:= stRoomDataPLC.bPirActive;
uiActLuxLevel_MB	:= stRoomDataPLC.uiActLuxLevel;

	//calculate BallastOnHours
	fbBallastOnHours(
		bEnableHourCount	:= bEnableHourCount,
		bPauseCount			:= fbLys.fbLightCtrl.bOffZone1,
		uiOnHours			:= uiBallastOnHours_MB,			//OnHours is updated here
		byOverflowCount		:= byOnHoursOverflowCount);


//Manage data for read/write for both PLC and MB registers
fbWriteSPLuxLevel(	nMaxValOut	:= uiMaxLuxLevel,
					nValIn1		:= uiSPLuxLevel_MB,		//nValIn1 takes priotity in case of download or restart
					nValIn2		:= stRoomDataPLC.uiSpLuxLevel,
					nValOut		=> uiLuxOn
				);


fbWritePirDelayTIme(	nMaxValOut	:= uiMaxPirOffMinutes,
						nValIn1		:= uiPirOffDelayTime_MB,		//nValIn1 takes priotity in case of download or restart
						nValIn2		:= stRoomDataPLC.uiPirOffDelayTime,
						nValOut		=> uiPirOffMinutes
					);
					

//Convert read/write modbus data to appropriate datatypes in PLC
fLuxOn	:= TO_REAL(uiLuxOn);			
tPIROff	:= TO_TIME(uiPirOffMinutes*udTimeScaling); //Time conversion defaults to ms

fLuxDim	:= TO_REAL(stRoomDataPLC.uiSpDimLuxLevel);			
tPIRDim	:= TO_TIME(stRoomDataPLC.uiPirDimDelayTime*udTimeScaling); //Time conversion defaults to ms
END_ACTION

ACTION A_Sensor:

fbSensor.ipCommunication := P_DALI_Background.arrfbKL6821Communication[Sensor_DALI_LINE_NUM];


fbSensor(
	byShrtAdr:= bySensorAddr,
	bInitialize:= bInitialize, 
	DALI_LINE_NUM:= Sensor_DALI_LINE_NUM, 
 	//bCancelHoldTimerOccupancy:= bCancelHoldTimerOccupancy, 
	stSensorSetup := stDaliSensorSetup,
	bInitErr=> bInitErr, 
	bInitDone=> bInitDone,
	stPirSensorData:= stPirSensorData, 
	arrSensorScales:= arrSensorScales);


(*
fbSensor(
	arrShrtAdr:= arrSensorAddr,
	bInitialize:= bInitialize, 
	DALI_LINE_NUM:= Sensor_DALI_LINE_NUM, 
 	//bCancelHoldTimerOccupancy:= bCancelHoldTimerOccupancy, 
	stSensorSetup := stDaliSensorSetup,
	arrInitErr=> arrInitErr, 
	arrInitDone=> arrInitDone,
	stPirSensorData:= stPirSensorData, 
	arrSensorScales:= arrSensorScales);
	*)
END_ACTION

END_PROGRAM

// ---- POUs/Alle_Rum/Rum_Med_DALI_Pir/Rum_4_211A/P_Rum_4_211A.TcPOU
PROGRAM P_Rum_4_211A
VAR
(*Rummet består af to lysgrupper - L1G3 og L2G3 - på to forskellige linjer
Begge grupper afhænger af samme PIR-input - pir-adr. 1 - på DALI-linje 2.
Derfor oprettes to adskilte reguleringer med samme PV. Dvs., at knapfunktion og pirfunktion forbliver den samme.
*)

	arrfbLysGruppe			: ARRAY [1..2] OF SH_Light.FB_Light_Type_A;
	arrstDaliSetupGruppe	: ARRAY [1..2] OF SH_Light.ST_DALI_RoomSetup := 
	
													[(	byShrtAdr_Prim := 12, 
														byGrpAdr_Prim := 3, 
														eMod_Prim := E_DALIAddressType.Group, 
														//byShrtAdr_Sec := 1, 
														//byGrpAdr_Sec := 1, 
														//eMod_Sec := E_DALIAddressType.Short, 
														//byShrtAdr_Supl := 1,
														//byGrpAdr_Supl := 1,
														//eMod_Supl := E_DALIADDRESSTYPE.Group,
														DALI_LINE_NUM_PRIM := arrDALI_LINE_NUM_LIGHT[1], 
														DALI_LINE_NUM_SEC := 0, //0 = ingen zonestyring/vinduerække
														DALI_LINE_NUM_SUPL := arrDALI_LINE_NUM_PENDANTS[1]),
														
													(	byShrtAdr_Prim := 7, 
														byGrpAdr_Prim := 3, 
														eMod_Prim := E_DALIAddressType.Group,
														//byShrtAdr_Sec := 1, 
														//byGrpAdr_Sec := 1, 
														//eMod_Sec := E_DALIAddressType.Short, 
														//byShrtAdr_Supl := 1,
														//byGrpAdr_Supl := 1,
														//eMod_Supl := E_DALIAddressType.Group, 
														DALI_LINE_NUM_PRIM := arrDALI_LINE_NUM_LIGHT[2], 
														DALI_LINE_NUM_SEC := 0, 
														DALI_LINE_NUM_SUPL := arrDALI_LINE_NUM_PENDANTS[2])];
														
	arrstLiveDataGruppe		: ARRAY [1..2] OF SH_Light.ST_LiveData;
	
	arrRunTuningGruppe: ARRAY[1..2] OF BOOL;
	
	bTopButtonZone1				: BOOL;
	bTopButtonZone1_Visu		: BOOL;
	bBottomButtonZone1			: BOOL;
	bBottomButtonZone1_Visu	: BOOL;
	bButtonZone2					: BOOL;
	bNeighborRoomsPir			: BOOL;
	fLuxOn								: REAL; 
	fLuxDim							: REAL;
	tPIRDim							: TIME;
	tPIROff							: TIME;
	fOffsetSec						: REAL := 20;
 

// Sensor Settings
	fbSensor					: SH_Light.FB_NIKO_P46xx_1Pcs;
	//fbSensor						: SH_Light.FB_NIKO_P46xx_2Pcs;
	bySensorAddr				: BYTE := 1;
	//arrSensorAddr				: ARRAY[1..2] OF BYTE := [1,2];
	bInitialize						: BOOL := TRUE;
	stDaliSensorSetup			: ST_DALI_NIKOP46SetupData;
	bInitErr							: BOOL;
	bInitDone						: BOOL;
	//arrInitErr						: ARRAY [1..2] OF BOOL;
	//arrInitDone					: ARRAY [1..2] OF BOOL;
	arrSensorScales				: ARRAY [1..10] OF SH_Light.ST_DALI_SensorScaleMode :=
																					[	(fMeassureMaxSensor := rMeassure_Zone11, fReadMaxSensor := rRead_Zone11),																		
																						9(())];
																																			
	bCancelHoldTimerOccupancy	: BOOL;
(*	eEventPriorityOccupancy		: E_DALIEventPriority := E_DALIEVENTPRIORITY.Middle;
	nHoldTimerOccupancy			: WORD := 5; // Value in s. 	
	nReportTimerOccupancy		: BYTE := 120; // Value in s, Preset manufacturer value
	nDeadtimeTimerOccupancy		: WORD := 100; // Value in ms, Predefined Value of DALI Standard
	bCancelHoldTimerOccupancy	: BOOL;
	nSensitivityOccupancy		: BYTE:= 3; //setting Sensivity (0..4) 0 (Off), 1 (Min), 2(Low), 3(High) and 4 (Max)

	bEnableLuxEvent				: BOOL;
	eEventPriorityBrightness	: E_DALIEventPriority := E_DALIEVENTPRIORITY.Middle;
	nDeadtimeTimerBrightness	: WORD := 1500; // Value in ms, Predefined Value of DALI Standard
	nHysteresisBrightness		: BYTE := 2; // Value in %
	nHysteresisMinBrightness	: BYTE := 10; // Absolute Value, depending on the manufacturer specific resolution
	nReportTimerBrightness		: BYTE := 120; // Value in s, Preset manufacturer value
*)


//ModbusComm setup
	
	fbWriteSPLuxLevel				: SH_Light.FB_TwoVal_SelectOne_RTrigChange;
	fbWritePirDelayTIme			: SH_Light.FB_TwoVal_SelectOne_RTrigChange;
	stRoomDataPLC					: SH_Light.ST_RoomDataPLC	:=	(	uiPirOffDelayTime	:= 30,
																										uiSpLuxLevel			:= 500,
																										uiPirDimDelayTime	:= 15,
																										uiSpDimLuxLevel		:= 200);
																
	fbBallastOnHours					: SH_Light.FB_CountOnHours;
	bEnableHourCount				: BOOL := TRUE;
	
	//Non-persistent modbus data
	bPirActive_MB					AT%MX76.0	: BOOL;				//bPirLys i gammel kode
	uiActLuxLevel_MB			AT%MB80		: UINT;				//intHMIAktueltLux i gammel kode
	uiActLightLevelPct_MB	AT%MB86		: UINT;				//intDALI_Gruppe1_Lysniveau i gammel kode
	
	//For Conversion
	uiPirOffMinutes						: UINT;
	udTimeScaling						: UDINT := 60000;
	uiLuxOn								: UINT;
	
	//max values checks
	uiMaxLuxLevel						: UINT := 1023;
	uiMaxPirOffMinutes					: UINT := 180;
	
END_VAR

VAR CONSTANT
	Sensor_DALI_LINE_NUM					: BYTE := 2;
	arrDALI_LINE_NUM_LIGHT				: ARRAY[1..2] OF BYTE := [1,2]; //korrekt rækkefølge nødvendig //rækkefølge og linje 
	arrDALI_LINE_NUM_PENDANTS	: ARRAY[1..2] OF BYTE := [0,0]; //korrekt rækkefølge nødvendig. 0 = ingen pendler
END_VAR

VAR PERSISTENT
	stPirSensorData										: SH_Light.ST_DALI_Sensor;
	arrstTuneDataGruppe								: ARRAY [1..2] OF SH_Light.ST_TuneData_EX;

	uiPirOffDelayTime_MB		AT%MB78	    : UINT;				//intHMI_Pir_SetValue i gammel kode
	uiSPLuxLevel_MB		    AT%MB82    	: UINT;				//intHMI_Lux_SetValue i gammel kode
	uiBallastOnHours_MB	    AT%MB90	    : UINT;				//dintHMILysbraendtimer1 i gammel kode
	byOnHoursOverflowCount			   				: BYTE;
END_VAR

A_Buttons();
A_LightCtrl();
A_ModbusComm();
A_Sensor();

ACTION A_Buttons:
bTopButtonZone1		:= GVL_EnOcean.strEnOceanSwitch_Rum_4_211A_Indgang.bT2_ON OR
									GVL_EnOcean.strEnOceanSwitch_Rum_4_211A_Ekstra.bT1_ON OR
									bTopButtonZone1_Visu;
bBottomButtonZone1	:= GVL_EnOcean.strEnOceanSwitch_Rum_4_211A_Indgang.bT2_OFF OR
									GVL_EnOcean.strEnOceanSwitch_Rum_4_211A_Ekstra.bT1_OFF OR
									bBottomButtonZone1_Visu;
END_ACTION

ACTION A_LightCtrl:
  
//gruppe L1G1
arrfbLysGruppe[1]( 
	nZoneID:= 1, 
	bButtonZone1:= bTopButtonZone1,
	bBottomButtonZone1 := bBottomButtonZone1,
	//bButtonZone2:= bButtonZone2,
	fLuxOn:= fLuxOn, 
	fLuxDim:= fLuxDim, 
	tPIRDim:= tPIRDim, 
	tPIROff:= tPIROff, 
	fOffsetSec:= fOffsetSec, 
	bReInit:= , 
	stDaliSetup:= arrstDaliSetupGruppe[1], 
	ipCommunication_Prim:= P_DALI_Background.arrfbKL6821Communication[arrDALI_LINE_NUM_LIGHT[1]], 
	//ipCommunication_Sec:= P_DALI_Background.arrfbKL6821Communication[arrDALI_LINE_NUM_LIGHT[1]], 
	//ipCommunication_Supl:= P_DALI_Background.arrfbKL6821Communication[arrDALI_LINE_NUM_PENDANTS[1]], 
	fMinOutputPowerLevelRoom:= 15, 
	fMaxOutputPowerLevelRoom:= 100, 
	nCycleTimeInMS:= SH_Light.DALI_Param.nPlcTaskCycleTimeInMS*nDimCmdCycleTimeFactor,   //Used only for dim. Factor=2 makes dimming smooth
	bRunTuning:= arrRunTuningGruppe[1], 
	bOccupiedRoom=> , 
	bError_Prim=> , 
	nError_Prim=> , 
	stTuneData:=arrstTuneDataGruppe[1] , 
	stPirSensorData:= stPirSensorData, 					//samme sensordata
	stLiveData:= arrstLiveDataGruppe[1]);

//gruppe 15	
arrfbLysGruppe[2]( 
	nZoneID:= 1, 
	bButtonZone1:= bTopButtonZone1,
	bBottomButtonZone1 := bBottomButtonZone1,
	//bButtonZone2:= bButtonZone2,
	fLuxOn:= fLuxOn, 
	fLuxDim:= fLuxDim, 
	tPIRDim:= tPIRDim, 
	tPIROff:= tPIROff, 
	fOffsetSec:= fOffsetSec, 
	bReInit:= , 
	stDaliSetup:= arrstDaliSetupGruppe[2], 
	ipCommunication_Prim:= P_DALI_Background.arrfbKL6821Communication[arrDALI_LINE_NUM_LIGHT[2]], 
	//ipCommunication_Sec:= P_DALI_Background.arrfbKL6821Communication[arrDALI_LINE_NUM_LIGHT[2]], 
	//ipCommunication_Supl:= P_DALI_Background.arrfbKL6821Communication[arrDALI_LINE_NUM_PENDANTS[2]], 
	fMinOutputPowerLevelRoom:= 15, 
	fMaxOutputPowerLevelRoom:= 100, 
	nCycleTimeInMS:= SH_Light.DALI_Param.nPlcTaskCycleTimeInMS*nDimCmdCycleTimeFactor,  //Used only for dim. Factor=2 makes dimming smooth
	bRunTuning:= arrRunTuningGruppe[2], 
	bOccupiedRoom=> , 
	bError_Prim=> , 
	nError_Prim=> , 
	stTuneData:=arrstTuneDataGruppe[2] , 
	stPirSensorData:= stPirSensorData, 					//samme sensordata
	stLiveData:= arrstLiveDataGruppe[2]);
END_ACTION

ACTION A_ModbusComm:
//Manage data for modbus communication

//Manage data for read-only in PLC
stRoomDataPLC.bPirActive			:= stPirSensorData.bPrc;
stRoomDataPLC.uiActLuxLevel			:= TO_UINT(TRUNC(stPirSensorData.fBrightness));
stRoomDataPLC.uiActLightLevelPct	:= TO_UINT(TRUNC(arrfbLysGruppe[1].fbBallast.fActlLgtLvl_Prim));
		//stRoomDataPLC.uiActLightLevelPct	:= TO_UINT(TRUNC(fbLys.fbBallast.fActlLgtLvl_Prim)); //if only one group light control
stRoomDataPLC.uiBallastOnHours		:= uiBallastOnHours_MB; //The calculation for BallastOnHours is stored directly to the MB register below


//Assign data for read-only to MB registers
bPirActive_MB		:= stRoomDataPLC.bPirActive;
uiActLuxLevel_MB	:= stRoomDataPLC.uiActLuxLevel;

	//calculate BallastOnHours
	fbBallastOnHours(
		bEnableHourCount	:= bEnableHourCount,
		bPauseCount			:= arrfbLysGruppe[1].fbLightCtrl.bOffZone1,
		uiOnHours			:= uiBallastOnHours_MB,			//OnHours is updated here
		byOverflowCount		:= byOnHoursOverflowCount);


//Manage data for read/write for both PLC and MB registers
fbWriteSPLuxLevel(	nMaxValOut	:= uiMaxLuxLevel,
					nValIn1		:= uiSPLuxLevel_MB,		//nValIn1 takes priotity in case of download or restart
					nValIn2		:= stRoomDataPLC.uiSpLuxLevel,
					nValOut		=> uiLuxOn
				);


fbWritePirDelayTIme(	nMaxValOut	:= uiMaxPirOffMinutes,
						nValIn1		:= uiPirOffDelayTime_MB,		//nValIn1 takes priotity in case of download or restart
						nValIn2		:= stRoomDataPLC.uiPirOffDelayTime,
						nValOut		=> uiPirOffMinutes
					);
					

//Convert read/write modbus data to appropriate datatypes in PLC
fLuxOn	:= TO_REAL(uiLuxOn);			
tPIROff	:= TO_TIME(uiPirOffMinutes*udTimeScaling); //Time conversion defaults to ms

fLuxDim	:= TO_REAL(stRoomDataPLC.uiSpDimLuxLevel);			
tPIRDim	:= TO_TIME(stRoomDataPLC.uiPirDimDelayTime*udTimeScaling); //Time conversion defaults to ms
END_ACTION

ACTION A_Sensor:

fbSensor.ipCommunication := P_DALI_Background.arrfbKL6821Communication[Sensor_DALI_LINE_NUM];

//only 1 sensor
fbSensor(
	byShrtAdr:= bySensorAddr,
	bInitialize:= bInitialize, 
	DALI_LINE_NUM:= Sensor_DALI_LINE_NUM, 
 	//bCancelHoldTimerOccupancy:= bCancelHoldTimerOccupancy, 
	stSensorSetup := stDaliSensorSetup,
	bInitErr=> bInitErr, 
	bInitDone=> bInitDone,
	stPirSensorData:= stPirSensorData, 
	arrSensorScales:= arrSensorScales);


//several sensors
(*	
fbSensor(
	arrShrtAdr:= arrSensorAddr,
	bInitialize:= bInitialize, 
	DALI_LINE_NUM:= Sensor_DALI_LINE_NUM, 
 	//bCancelHoldTimerOccupancy:= bCancelHoldTimerOccupancy, 
	stSensorSetup := stDaliSensorSetup,
	arrInitErr=> arrInitErr, 
	arrInitDone=> arrInitDone,
	stPirSensorData:= stPirSensorData, 
	arrSensorScales:= arrSensorScales);
	*)
END_ACTION

END_PROGRAM

// ---- POUs/Alle_Rum/Rum_Med_DALI_Pir/Rum_4_213_Og_4_215_Foldedoer/P_Rum_4_213.TcPOU
PROGRAM P_Rum_4_213
VAR
(*Rummet består af to lysgrupper - L1G4 og L2G4 - på to forskellige linjer
Begge grupper afhænger af samme PIR-input - pir-adr. 3, 4, 6 og 7 - på DALI-linje 2.
Derfor oprettes to adskilte reguleringer med samme PV.
Yderligere logik for knapfunktion og pirsignaler håndteres i program for foldedør 
*)

	arrfbLysGruppe			: ARRAY [1..2] OF SH_Light.FB_Light_Type_A;
	arrstDaliSetupGruppe	: ARRAY [1..2] OF SH_Light.ST_DALI_RoomSetup := 
	
													[(	byShrtAdr_Prim := 15, 
														byGrpAdr_Prim := 4, 
														eMod_Prim := E_DALIAddressType.Group, 
														//byShrtAdr_Sec := 1, 
														//byGrpAdr_Sec := 1, 
														//eMod_Sec := E_DALIAddressType.Short, 
														byShrtAdr_Supl := 15,
														//byGrpAdr_Supl := 1,
														eMod_Supl := E_DALIADDRESSTYPE.Short,
														DALI_LINE_NUM_PRIM := arrDALI_LINE_NUM_LIGHT[1], 
														DALI_LINE_NUM_SEC := 0, //0 = ingen zonestyring/vinduerække
														DALI_LINE_NUM_SUPL := arrDALI_LINE_NUM_PENDANTS[1]),
														
													(	byShrtAdr_Prim := 11, 
														byGrpAdr_Prim := 4, 
														eMod_Prim := E_DALIAddressType.Group,
														//byShrtAdr_Sec := 1, 
														//byGrpAdr_Sec := 1, 
														//eMod_Sec := E_DALIAddressType.Short, 
														//byShrtAdr_Supl := 1,
														//byGrpAdr_Supl := 1,
														//eMod_Supl := E_DALIAddressType.Group, 
														DALI_LINE_NUM_PRIM := arrDALI_LINE_NUM_LIGHT[2], 
														DALI_LINE_NUM_SEC := 0, 
														DALI_LINE_NUM_SUPL := arrDALI_LINE_NUM_PENDANTS[2])];
														
	arrstLiveDataGruppe		: ARRAY [1..2] OF SH_Light.ST_LiveData;
	
	arrRunTuningGruppe: ARRAY[1..2] OF BOOL;
	
	bTopButtonZone1				: BOOL;
	bTopButtonZone1_Visu		: BOOL;
	bBottomButtonZone1			: BOOL;
	bBottomButtonZone1_Visu	: BOOL;
	bButtonZone2					: BOOL;
	bNeighborRoomsPir			: BOOL;
	fLuxOn								: REAL; 
	fLuxDim							: REAL;
	tPIRDim							: TIME;
	tPIROff							: TIME;
	fOffsetSec						: REAL := 20;
 

// Sensor Settings
	//fbSensor					: SH_Light.FB_NIKO_P46xx_1Pcs;
	fbSensor						: SH_Light.FB_NIKO_P46xx_4Pcs;
	//bySensorAddr				: BYTE := 1;
	arrSensorAddr				: ARRAY[1..4] OF BYTE := [3,4,6,7];
	bInitialize						: BOOL := TRUE;
	stDaliSensorSetup			: ST_DALI_NIKOP46SetupData;
	//bInitErr							: BOOL;
	//bInitDone						: BOOL;
	arrInitErr						: ARRAY [1..4] OF BOOL;
	arrInitDone					: ARRAY [1..4] OF BOOL;
	arrSensorScales				: ARRAY [1..10] OF SH_Light.ST_DALI_SensorScaleMode :=
																					[	(fMeassureMaxSensor := rMeassure_Zone5, fReadMaxSensor := rRead_Zone5),
																						(fMeassureMaxSensor := rMeassure_Zone5, fReadMaxSensor := rRead_Zone5),
																						(fMeassureMaxSensor := rMeassure_Zone5, fReadMaxSensor := rRead_Zone5),
																						(fMeassureMaxSensor := rMeassure_Zone5, fReadMaxSensor := rRead_Zone5),																	
																						6(())];
																																			
	bCancelHoldTimerOccupancy	: BOOL;
(*	eEventPriorityOccupancy		: E_DALIEventPriority := E_DALIEVENTPRIORITY.Middle;
	nHoldTimerOccupancy			: WORD := 5; // Value in s. 	
	nReportTimerOccupancy		: BYTE := 120; // Value in s, Preset manufacturer value
	nDeadtimeTimerOccupancy		: WORD := 100; // Value in ms, Predefined Value of DALI Standard
	bCancelHoldTimerOccupancy	: BOOL;
	nSensitivityOccupancy		: BYTE:= 3; //setting Sensivity (0..4) 0 (Off), 1 (Min), 2(Low), 3(High) and 4 (Max)

	bEnableLuxEvent				: BOOL;
	eEventPriorityBrightness	: E_DALIEventPriority := E_DALIEVENTPRIORITY.Middle;
	nDeadtimeTimerBrightness	: WORD := 1500; // Value in ms, Predefined Value of DALI Standard
	nHysteresisBrightness		: BYTE := 2; // Value in %
	nHysteresisMinBrightness	: BYTE := 10; // Absolute Value, depending on the manufacturer specific resolution
	nReportTimerBrightness		: BYTE := 120; // Value in s, Preset manufacturer value
*)


//ModbusComm setup
	
	fbWriteSPLuxLevel				: SH_Light.FB_TwoVal_SelectOne_RTrigChange;
	fbWritePirDelayTIme			: SH_Light.FB_TwoVal_SelectOne_RTrigChange;
	stRoomDataPLC					: SH_Light.ST_RoomDataPLC	:=	(	uiPirOffDelayTime	:= 30,
																										uiSpLuxLevel			:= 500,
																										uiPirDimDelayTime	:= 15,
																										uiSpDimLuxLevel		:= 200);
																
	fbBallastOnHours					: SH_Light.FB_CountOnHours;
	bEnableHourCount				: BOOL := TRUE;
	
	//Non-persistent modbus data
	bPirActive_MB					AT%MX120.0	: BOOL;				//bPirLys i gammel kode
	uiActLuxLevel_MB			AT%MB124		: UINT;				//intHMIAktueltLux i gammel kode
	uiActLightLevelPct_MB	AT%MB132		: UINT;				//intDALI_Gruppe1_Lysniveau i gammel kode
	
	//For Conversion
	uiPirOffMinutes						: UINT;
	udTimeScaling						: UDINT := 60000;
	uiLuxOn								: UINT;
	
	//max values checks
	uiMaxLuxLevel						: UINT := 1023;
	uiMaxPirOffMinutes					: UINT := 180;
	
END_VAR

VAR CONSTANT
	Sensor_DALI_LINE_NUM					: BYTE := 2;
	arrDALI_LINE_NUM_LIGHT				: ARRAY[1..2] OF BYTE := [1,2]; //korrekt rækkefølge nødvendig //rækkefølge og linje 
	arrDALI_LINE_NUM_PENDANTS	: ARRAY[1..2] OF BYTE := [2,0]; //korrekt rækkefølge nødvendig. 0 = ingen pendler
END_VAR

VAR PERSISTENT
	stPirSensorData										: SH_Light.ST_DALI_Sensor;
	arrstTuneDataGruppe								: ARRAY [1..2] OF SH_Light.ST_TuneData_EX;

	uiPirOffDelayTime_MB		AT%MB122	    : UINT;				//intHMI_Pir_SetValue i gammel kode
	uiSPLuxLevel_MB		    AT%MB128    	: UINT;				//intHMI_Lux_SetValue i gammel kode
	uiBallastOnHours_MB	    AT%MB136	    : UINT;				//dintHMILysbraendtimer1 i gammel kode
	byOnHoursOverflowCount			   				: BYTE;
END_VAR

A_Buttons();
A_LightCtrl();
A_ModbusComm();
A_Sensor();

ACTION A_Buttons:
//Yderligere Logik for knapper håndteres i P_Foldedoer_4_213

bTopButtonZone1		:= P_Foldedoer_4_213.arrTopButtonZone1Comb[1] OR bTopButtonZone1_Visu;
bBottomButtonZone1	:= P_Foldedoer_4_213.arrBottomButtonZone1Comb[1] OR bBottomButtonZone1_Visu;

bButtonZone2			:= GVL_EnOcean.strEnOceanSwitch_Rum_4_213_Pendler.bT2_ON OR GVL_EnOcean.strEnOceanSwitch_Rum_4_213_Pendler.bT2_OFF;
END_ACTION

ACTION A_LightCtrl:
  
//gruppe L1G1
arrfbLysGruppe[1]( 
	nZoneID:= 1, 
	bButtonZone1:= bTopButtonZone1,
	bBottomButtonZone1 := bBottomButtonZone1,
	bButtonZone2:= bButtonZone2,
	fLuxOn:= fLuxOn, 
	fLuxDim:= fLuxDim, 
	tPIRDim:= tPIRDim, 
	tPIROff:= tPIROff, 
	fOffsetSec:= fOffsetSec, 
	bReInit:= , 
	stDaliSetup:= arrstDaliSetupGruppe[1], 
	ipCommunication_Prim:= P_DALI_Background.arrfbKL6821Communication[arrDALI_LINE_NUM_LIGHT[1]], 
	//ipCommunication_Sec:= P_DALI_Background.arrfbKL6821Communication[arrDALI_LINE_NUM_LIGHT[1]], 
	ipCommunication_Supl:= P_DALI_Background.arrfbKL6821Communication[arrDALI_LINE_NUM_PENDANTS[1]], 
	fMinOutputPowerLevelRoom:= 15, 
	fMaxOutputPowerLevelRoom:= 100, 
	nCycleTimeInMS:= SH_Light.DALI_Param.nPlcTaskCycleTimeInMS*nDimCmdCycleTimeFactor,   //Used only for dim. Factor=2 makes dimming smooth
	bRunTuning:= arrRunTuningGruppe[1], 
	bOccupiedRoom=> , 
	bError_Prim=> , 
	nError_Prim=> , 
	stTuneData:=arrstTuneDataGruppe[1] , 
	stPirSensorData:= P_Foldedoer_4_213.arrstPirSensorDataComb[1], 					//samme sensordata
	stLiveData:= arrstLiveDataGruppe[1]);

//gruppe 15	
arrfbLysGruppe[2]( 
	nZoneID:= 1, 
	bButtonZone1:= bTopButtonZone1,
	bBottomButtonZone1 := bBottomButtonZone1,
	//bButtonZone2:= bButtonZone2,
	fLuxOn:= fLuxOn, 
	fLuxDim:= fLuxDim, 
	tPIRDim:= tPIRDim, 
	tPIROff:= tPIROff, 
	fOffsetSec:= fOffsetSec, 
	bReInit:= , 
	stDaliSetup:= arrstDaliSetupGruppe[2], 
	ipCommunication_Prim:= P_DALI_Background.arrfbKL6821Communication[arrDALI_LINE_NUM_LIGHT[2]], 
	//ipCommunication_Sec:= P_DALI_Background.arrfbKL6821Communication[arrDALI_LINE_NUM_LIGHT[2]], 
	//ipCommunication_Supl:= P_DALI_Background.arrfbKL6821Communication[arrDALI_LINE_NUM_PENDANTS[2]], 
	fMinOutputPowerLevelRoom:= 15, 
	fMaxOutputPowerLevelRoom:= 100, 
	nCycleTimeInMS:= SH_Light.DALI_Param.nPlcTaskCycleTimeInMS*nDimCmdCycleTimeFactor,  //Used only for dim. Factor=2 makes dimming smooth
	bRunTuning:= arrRunTuningGruppe[2], 
	bOccupiedRoom=> , 
	bError_Prim=> , 
	nError_Prim=> , 
	stTuneData:=arrstTuneDataGruppe[2] , 
	stPirSensorData:= P_Foldedoer_4_213.arrstPirSensorDataComb[1], 					//samme sensordata
	stLiveData:= arrstLiveDataGruppe[2]);
END_ACTION

ACTION A_ModbusComm:
//Manage data for modbus communication

//Manage data for read-only in PLC
stRoomDataPLC.bPirActive			:= stPirSensorData.bPrc;
stRoomDataPLC.uiActLuxLevel			:= TO_UINT(TRUNC(stPirSensorData.fBrightness));
stRoomDataPLC.uiActLightLevelPct	:= TO_UINT(TRUNC(arrfbLysGruppe[1].fbBallast.fActlLgtLvl_Prim));
		//stRoomDataPLC.uiActLightLevelPct	:= TO_UINT(TRUNC(fbLys.fbBallast.fActlLgtLvl_Prim)); //if only one group light control
stRoomDataPLC.uiBallastOnHours		:= uiBallastOnHours_MB; //The calculation for BallastOnHours is stored directly to the MB register below


//Assign data for read-only to MB registers
bPirActive_MB		:= stRoomDataPLC.bPirActive;
uiActLuxLevel_MB	:= stRoomDataPLC.uiActLuxLevel;

	//calculate BallastOnHours
	fbBallastOnHours(
		bEnableHourCount	:= bEnableHourCount,
		bPauseCount			:= arrfbLysGruppe[1].fbLightCtrl.bOffZone1,
		uiOnHours			:= uiBallastOnHours_MB,			//OnHours is updated here
		byOverflowCount		:= byOnHoursOverflowCount);


//Manage data for read/write for both PLC and MB registers
fbWriteSPLuxLevel(	nMaxValOut	:= uiMaxLuxLevel,
					nValIn1		:= uiSPLuxLevel_MB,		//nValIn1 takes priotity in case of download or restart
					nValIn2		:= stRoomDataPLC.uiSpLuxLevel,
					nValOut		=> uiLuxOn
				);


fbWritePirDelayTIme(	nMaxValOut	:= uiMaxPirOffMinutes,
						nValIn1		:= uiPirOffDelayTime_MB,		//nValIn1 takes priotity in case of download or restart
						nValIn2		:= stRoomDataPLC.uiPirOffDelayTime,
						nValOut		=> uiPirOffMinutes
					);
					

//Convert read/write modbus data to appropriate datatypes in PLC
fLuxOn	:= TO_REAL(uiLuxOn);			
tPIROff	:= TO_TIME(uiPirOffMinutes*udTimeScaling); //Time conversion defaults to ms

fLuxDim	:= TO_REAL(stRoomDataPLC.uiSpDimLuxLevel);			
tPIRDim	:= TO_TIME(stRoomDataPLC.uiPirDimDelayTime*udTimeScaling); //Time conversion defaults to ms
END_ACTION

ACTION A_Sensor:

fbSensor.ipCommunication := P_DALI_Background.arrfbKL6821Communication[Sensor_DALI_LINE_NUM];

//only 1 sensor
(*
fbSensor(
	byShrtAdr:= bySensorAddr,
	bInitialize:= bInitialize, 
	DALI_LINE_NUM:= Sensor_DALI_LINE_NUM, 
 	//bCancelHoldTimerOccupancy:= bCancelHoldTimerOccupancy, 
	stSensorSetup := stDaliSensorSetup,
	bInitErr=> bInitErr, 
	bInitDone=> bInitDone,
	stPirSensorData:= stPirSensorData, 
	arrSensorScales:= arrSensorScales);
*)

//several sensors	
fbSensor(
	arrShrtAdr:= arrSensorAddr,
	bInitialize:= bInitialize, 
	DALI_LINE_NUM:= Sensor_DALI_LINE_NUM, 
 	//bCancelHoldTimerOccupancy:= bCancelHoldTimerOccupancy, 
	stSensorSetup := stDaliSensorSetup,
	arrInitErr=> arrInitErr, 
	arrInitDone=> arrInitDone,
	stPirSensorData:= P_Foldedoer_4_213.arrstPirSensorData[1], 
	arrSensorScales:= arrSensorScales);
	
	stPirSensorData := P_Foldedoer_4_213.arrstPirSensorData[1]; //For at holde samme navngivning i A_ModbusComm
END_ACTION

END_PROGRAM

// ---- POUs/Alle_Rum/Rum_Med_DALI_Pir/Rum_4_213_Og_4_215_Foldedoer/P_Foldedoer_4_213.TcPOU
PROGRAM P_Foldedoer_4_213
(*
Rummene er delt af en foldedør med dørkontakt i rum 4.213. Når dørkontakt aktiveres behandles de to rum som ét rum:
	- Senorinput sammensættes, således de to reguleringer har samme PV.
	- Knapfunktion sammensættes, således alle knapper kan benyttes for hele rummet.
Sammensætning af sensorinput foregår i FB_FoldingDoor.A_SensorLogic (SH_Light)
Sammensætning af knapfunktion foregår i FB_FoldingDoor.A_ButtonLogic (SH_Light)

Rækkefølge i arrays: [1, 2] = [*rum 4.213*, *rum 4.215*]
*)
VAR
	bFoldingDoorOpen 		AT %I*	: BOOL;
	
	arrTopButtonZone1						: ARRAY[1..2] OF BOOL; //Fra GVL_EnOcean
	arrBottomButtonZone1					: ARRAY[1..2] OF BOOL; //Fra GVL_EnOcean
	arrTopButtonZone1Comb				: ARRAY[1..2] OF BOOL; //Til A_Buttons
	arrBottomButtonZone1Comb			: ARRAY[1..2] OF BOOL; //Til A_Buttons
	
	arrstPirSensorData						: ARRAY[1..2] OF SH_Light.ST_DALI_Sensor; //VAR_IN_OUT til og fra sensorer
	arrstPirSensorDataComb				: ARRAY[1..2] OF SH_Light.ST_DALI_Sensor; //VAR_IN_OUT til og fra LightCtrl
	
	fbFoldingDoor								: SH_Light.FB_FoldingDoor;
END_VAR

arrTopButtonZone1[1]		:= GVL_EnOcean.strEnOceanSwitch_Rum_4_213_Indgang.bT2_ON;
arrBottomButtonZone1[1]	:= GVL_EnOcean.strEnOceanSwitch_Rum_4_213_Indgang.bT2_OFF;
arrTopButtonZone1[2]		:= GVL_EnOcean.strEnOceanSwitch_Rum_4_215.bT2_ON;
arrBottomButtonZone1[2]	:= GVL_EnOcean.strEnOceanSwitch_Rum_4_215.bT2_OFF;

fbFoldingDoor(
	bFoldingDoorOpen 				:= bFoldingDoorOpen,
	arrTopButtonZone1 				:= arrTopButtonZone1,
	arrBottomButtonZone1			:= arrBottomButtonZone1,
	arrstPirSensorData				:= arrstPirSensorData,
	arrstPirSensorDataComb		:= arrstPirSensorDataComb,
	arrTopButtonZone1Comb		=> arrTopButtonZone1Comb,
	arrBottomButtonZone1Comb	=> arrBottomButtonZone1Comb);
(*
A_ButtonLogic();
A_SensorLogic();
*)

ACTION A_ButtonLogic:
arrTopButtonZone1[1] := GVL_EnOcean.strEnOceanSwitch_Rum_4_217.bT2_OFF;
arrBottomButtonZone1[1] := GVL_EnOcean.strEnOceanSwitch_Rum_4_217.bT2_ON;
arrTopButtonZone1[2] := GVL_EnOcean.strEnOceanSwitch_Rum_4_219.bT2_ON;
arrBottomButtonZone1[2] := GVL_EnOcean.strEnOceanSwitch_Rum_4_219.bT2_OFF;

IF bFoldingDoorOpen THEN
	arrTopButtonZone1Comb[1] := arrTopButtonZone1[1] OR arrTopButtonZone1[2];
	arrTopButtonZone1Comb[2] := arrTopButtonZone1Comb[1];
	arrBottomButtonZone1Comb[1] := arrBottomButtonZone1[1] OR arrBottomButtonZone1[2];
	arrBottomButtonZone1Comb[2] := arrBottomButtonZone1Comb[1];
ELSE
	arrTopButtonZone1Comb := arrTopButtonZone1;
	arrBottomButtonZone1Comb := arrBottomButtonZone1;
END_IF
END_ACTION

ACTION A_SensorLogic:
IF bFoldingDoorOpen THEN
	//Input fra sensorer samles
	arrstPirSensorDataComb[1].fBrightness			:= MIN(arrstPirSensorData[1].fBrightness, arrstPirSensorData[2].fBrightness);
	arrstPirSensorDataComb[1].bPrc					:= arrstPirSensorData[1].bPrc OR arrstPirSensorData[2].bPrc;
	arrstPirSensorDataComb[1].bBrightnessRead	:= arrstPirSensorData[1].bBrightnessRead OR arrstPirSensorData[2].bBrightnessRead;
	arrstPirSensorDataComb[2].fBrightness			:= arrstPirSensorDataComb[1].fBrightness;
	arrstPirSensorDataComb[2].bPrc					:= arrstPirSensorDataComb[1].bPrc;
	arrstPirSensorDataComb[2].bBrightnessRead	:= arrstPirSensorDataComb[1].bBrightnessRead;

	//Output til sensorer fordeles
	IF arrstPirSensorDataComb[1].bQueryBrightness OR arrstPirSensorDataComb[2].bQueryBrightness THEN
		arrstPirSensorData[1].bQueryBrightness := TRUE;
		arrstPirSensorData[2].bQueryBrightness := TRUE;
	ELSE
		arrstPirSensorData[1].bQueryBrightness := FALSE;
		arrstPirSensorData[2].bQueryBrightness := FALSE;
	END_IF
ELSE
	//Input fra sensorer samles uden ændring
	arrstPirSensorDataComb[1].fBrightness			:= arrstPirSensorData[1].fBrightness;
	arrstPirSensorDataComb[1].bPrc					:= arrstPirSensorData[1].bPrc;
	arrstPirSensorDataComb[1].bBrightnessRead	:= arrstPirSensorData[1].bBrightnessRead;
	arrstPirSensorDataComb[2].fBrightness			:= arrstPirSensorData[2].fBrightness;
	arrstPirSensorDataComb[2].bPrc					:= arrstPirSensorData[2].bPrc;
	arrstPirSensorDataComb[2].bBrightnessRead := arrstPirSensorData[2].bBrightnessRead;
	
	//Output til sensorer fordeles uden ændring
	IF arrstPirSensorDataComb[1].bQueryBrightness THEN
		arrstPirSensorData[1].bQueryBrightness := TRUE;
	ELSE
		arrstPirSensorData[1].bQueryBrightness := FALSE;
	END_IF
	IF arrstPirSensorDataComb[2].bQueryBrightness THEN
		arrstPirSensorData[2].bQueryBrightness := TRUE;
	ELSE
		arrstPirSensorData[2].bQueryBrightness := FALSE;
	END_IF
END_IF
END_ACTION

END_PROGRAM

// ---- POUs/Alle_Rum/Gange/Gang_4_211/P_Gang_4_211.TcPOU
PROGRAM P_Gang_4_211
VAR
(*Gangen består af en lysgruppe og et ekstra armatur - L2G2 og L1S14 - på to forskellige linjer
Både gruppen og ekstra armatur afhænger af samme PIR-input - pir-adr. 2 - på DALI-linje 2.
Derfor oprettes to adskilte reguleringer med samme PV. Dvs., at knapfunktion og pirfunktion forbliver den samme.
*)

	arrfbLysGruppe			: ARRAY [1..2] OF SH_Light.FB_Light_Type_B;
	arrstDaliSetupGruppe	: ARRAY [1..2] OF SH_Light.ST_DALI_RoomSetup := 
	
													[(	byShrtAdr_Prim := 14, 
														//byGrpAdr_Prim := 1, 
														eMod_Prim := E_DALIAddressType.Short, 
														//byShrtAdr_Sec := 1, 
														//byGrpAdr_Sec := 1, 
														//eMod_Sec := E_DALIAddressType.Short, 
														//byShrtAdr_Supl := 1,
														//byGrpAdr_Supl := 1,
														//eMod_Supl := E_DALIADDRESSTYPE.Group,
														DALI_LINE_NUM_PRIM := arrDALI_LINE_NUM_LIGHT[1], 
														DALI_LINE_NUM_SEC := 0, //0 = ingen zonestyring/vinduerække
														DALI_LINE_NUM_SUPL := arrDALI_LINE_NUM_PENDANTS[1]),
														
													(	byShrtAdr_Prim := 9, 
														byGrpAdr_Prim := 2, 
														eMod_Prim := E_DALIAddressType.Group,
														//byShrtAdr_Sec := 1, 
														//byGrpAdr_Sec := 1, 
														//eMod_Sec := E_DALIAddressType.Short, 
														//byShrtAdr_Supl := 1,
														//byGrpAdr_Supl := 1,
														//eMod_Supl := E_DALIAddressType.Group, 
														DALI_LINE_NUM_PRIM := arrDALI_LINE_NUM_LIGHT[2], 
														DALI_LINE_NUM_SEC := 0, 
														DALI_LINE_NUM_SUPL := arrDALI_LINE_NUM_PENDANTS[2])];
														
	arrstLiveDataGruppe		: ARRAY [1..2] OF SH_Light.ST_LiveData;
	
	arrRunTuningGruppe: ARRAY[1..2] OF BOOL;
	
	bTopButtonZone1				: BOOL;
	bTopButtonZone1_Visu		: BOOL;
	bBottomButtonZone1			: BOOL;
	bBottomButtonZone1_Visu	: BOOL;
	bButtonZone2					: BOOL;
	bNeighborRoomsPir			: BOOL;
	fLuxOn								: REAL; 
	fLuxDim							: REAL;
	tPIRDim							: TIME;
	tPIROff							: TIME;
	fOffsetSec						: REAL := 20;
 

// Sensor Settings
	fbSensor					: SH_Light.FB_NIKO_P46xx_1Pcs;
	//fbSensor						: SH_Light.FB_NIKO_P46xx_2Pcs;
	bySensorAddr				: BYTE := 2;
	//arrSensorAddr				: ARRAY[1..2] OF BYTE := [1,2];
	bInitialize						: BOOL := TRUE;
	stDaliSensorSetup			: ST_DALI_NIKOP46SetupData;
	bInitErr							: BOOL;
	bInitDone						: BOOL;
	//arrInitErr						: ARRAY [1..2] OF BOOL;
	//arrInitDone					: ARRAY [1..2] OF BOOL;
	arrSensorScales				: ARRAY [1..10] OF SH_Light.ST_DALI_SensorScaleMode :=
																					[	(fMeassureMaxSensor := rMeassure_Zone10, fReadMaxSensor := rRead_Zone10),																		
																						9(())];
																																			
	bCancelHoldTimerOccupancy	: BOOL;
(*	eEventPriorityOccupancy		: E_DALIEventPriority := E_DALIEVENTPRIORITY.Middle;
	nHoldTimerOccupancy			: WORD := 5; // Value in s. 	
	nReportTimerOccupancy		: BYTE := 120; // Value in s, Preset manufacturer value
	nDeadtimeTimerOccupancy		: WORD := 100; // Value in ms, Predefined Value of DALI Standard
	bCancelHoldTimerOccupancy	: BOOL;
	nSensitivityOccupancy		: BYTE:= 3; //setting Sensivity (0..4) 0 (Off), 1 (Min), 2(Low), 3(High) and 4 (Max)

	bEnableLuxEvent				: BOOL;
	eEventPriorityBrightness	: E_DALIEventPriority := E_DALIEVENTPRIORITY.Middle;
	nDeadtimeTimerBrightness	: WORD := 1500; // Value in ms, Predefined Value of DALI Standard
	nHysteresisBrightness		: BYTE := 2; // Value in %
	nHysteresisMinBrightness	: BYTE := 10; // Absolute Value, depending on the manufacturer specific resolution
	nReportTimerBrightness		: BYTE := 120; // Value in s, Preset manufacturer value
*)


//ModbusComm setup
	
	fbWriteSPLuxLevel				: SH_Light.FB_TwoVal_SelectOne_RTrigChange;
	fbWritePirDelayTIme			: SH_Light.FB_TwoVal_SelectOne_RTrigChange;
	stRoomDataPLC					: SH_Light.ST_RoomDataPLC	:=	(	uiPirOffDelayTime	:= 30,
																										uiSpLuxLevel			:= 500,
																										uiPirDimDelayTime	:= 15,
																										uiSpDimLuxLevel		:= 200);
																
	fbBallastOnHours					: SH_Light.FB_CountOnHours;
	bEnableHourCount				: BOOL := TRUE;
	
	//Non-persistent modbus data
	bPirActive_MB					AT%MX168.0	: BOOL;				//bPirLys i gammel kode
	uiActLuxLevel_MB			AT%MB176		: UINT;				//intHMIAktueltLux i gammel kode
	uiActLightLevelPct_MB	AT%MB172		: UINT;				//intDALI_Gruppe1_Lysniveau i gammel kode
	
	//For Conversion
	uiPirOffMinutes						: UINT;
	udTimeScaling						: UDINT := 60000;
	uiLuxOn								: UINT;
	
	//max values checks
	uiMaxLuxLevel						: UINT := 1023;
	uiMaxPirOffMinutes				: UINT := 180;
	
END_VAR

VAR CONSTANT
	Sensor_DALI_LINE_NUM					: BYTE := 2;
	arrDALI_LINE_NUM_LIGHT				: ARRAY[1..2] OF BYTE := [1,2]; //korrekt rækkefølge nødvendig //rækkefølge og linje 
	arrDALI_LINE_NUM_PENDANTS	: ARRAY[1..2] OF BYTE := [0,0]; //korrekt rækkefølge nødvendig. 0 = ingen pendler
END_VAR

VAR PERSISTENT
	stPirSensorData										: SH_Light.ST_DALI_Sensor;
	arrstTuneDataGruppe								: ARRAY [1..2] OF SH_Light.ST_TuneData_EX;

	uiPirOffDelayTime_MB		AT%MB170	    : UINT;				//intHMI_Pir_SetValue i gammel kode
	uiSPLuxLevel_MB		    AT%MB178    	: UINT;				//intHMI_Lux_SetValue i gammel kode
	uiBallastOnHours_MB	    AT%MB174	    : UINT;				//dintHMILysbraendtimer1 i gammel kode
	byOnHoursOverflowCount			   				: BYTE;
END_VAR

A_Buttons();
A_LightCtrl();
A_ModbusComm();
A_Sensor();

ACTION A_Buttons:
bTopButtonZone1		:= GVL_EnOcean.strEnOceanSwitch_Gang_4_211_Indgang.bT2_ON OR
									GVL_EnOcean.strEnOceanSwitch_Gang_4_211_Ekstra.bT1_ON OR
									bTopButtonZone1_Visu;
bBottomButtonZone1	:= GVL_EnOcean.strEnOceanSwitch_Gang_4_211_Indgang.bT2_OFF OR
									GVL_EnOcean.strEnOceanSwitch_Gang_4_211_Ekstra.bT1_OFF OR
									bBottomButtonZone1_Visu;
END_ACTION

ACTION A_LightCtrl:
  bNeighborRoomsPir	 :=		P_Rum_4_211A.stPirSensorData.bPrc;
  
//L1S14
arrfbLysGruppe[1]( 
	nZoneID:= 1, 
	bButtonZone1:= bTopButtonZone1,
	bBottomButtonZone1 := bBottomButtonZone1,
	//bButtonZone2:= bButtonZone2,
	bNeighborRoomsPir := bNeighborRoomsPir,
	fLuxOn:= fLuxOn, 
	fLuxDim:= fLuxDim, 
	tPIRDim:= tPIRDim, 
	tPIROff:= tPIROff, 
	fOffsetSec:= fOffsetSec, 
	bReInit:= , 
	stDaliSetup:= arrstDaliSetupGruppe[1], 
	ipCommunication_Prim:= P_DALI_Background.arrfbKL6821Communication[arrDALI_LINE_NUM_LIGHT[1]], 
	//ipCommunication_Sec:= P_DALI_Background.arrfbKL6821Communication[arrDALI_LINE_NUM_LIGHT[1]], 
	//ipCommunication_Supl:= P_DALI_Background.arrfbKL6821Communication[arrDALI_LINE_NUM_PENDANTS[1]], 
	fMinOutputPowerLevelRoom:= 15, 
	fMaxOutputPowerLevelRoom:= 100, 
	nCycleTimeInMS:= SH_Light.DALI_Param.nPlcTaskCycleTimeInMS*nDimCmdCycleTimeFactor,   //Used only for dim. Factor=2 makes dimming smooth
	bRunTuning:= arrRunTuningGruppe[1], 
	bOccupiedRoom=> , 
	bError_Prim=> , 
	nError_Prim=> , 
	stTuneData:=arrstTuneDataGruppe[1] , 
	stPirSensorData:= stPirSensorData, 					//samme sensordata
	stLiveData:= arrstLiveDataGruppe[1]);

